LIN {X 0,Y 364.12,Z 423.241,A -85,B 0,C 180,E1 -13065.677,E2 -13065.677} C_VEL
LIN {X 0,Y 365.365,Z 412.607,A -85,B 0,C 180,E1 -13066.914,E2 -13066.914} C_VEL
LIN {X 0,Y 366.671,Z 400.866,A -85,B 0,C 180,E1 -13068.003,E2 -13068.003} C_VEL
LIN {X 0,Y 367.855,Z 388.491,A -85,B 0,C 180,E1 -13068.88,E2 -13068.88} C_VEL
LIN {X 0,Y 368.998,Z 374.969,A -85,B 0,C 180,E1 -13069.578,E2 -13069.578} C_VEL
LIN {X 0,Y 369.706,Z 361.353,A -85,B 0,C 180,E1 -13070.041,E2 -13070.041} C_VEL
LIN {X 0,Y 371.251,Z 294.99,A -85,B 0,C 180,E1 -13071.529,E2 -13071.529} C_VEL
LIN {X 0,Y 368.499,Z 273.063,A -85,B 0,C 180,E1 -13072.273,E2 -13072.273} C_VEL
LIN {X 0,Y 365.195,Z 254.41,A -85,B 0,C 180,E1 -13073,E2 -13073} C_VEL
LIN {X 0,Y 364.953,Z 252.892,A -85,B 0,C 180,E1 -13073.063,E2 -13073.063} C_VEL
LIN {X 0,Y 366.552,Z 235.571,A -85,B 0,C 180,E1 -13076.473,E2 -13076.473} C_VEL
LIN {X 0,Y 366.814,Z 231.096,A -85,B 0,C 180,E1 -13077.376,E2 -13077.376} C_VEL
LIN {X 0,Y 364.611,Z 220.318,A -85,B 0,C 180,E1 -13079.843,E2 -13079.843} C_VEL
LIN {X 0,Y 361.857,Z 209.412,A -85,B 0,C 180,E1 -13082.53,E2 -13082.53} C_VEL
LIN {X 0,Y 361.868,Z 209.408,A -85,B 0,C 180,E1 -13085.636,E2 -13085.636} C_VEL
LIN {X 0,Y 361.826,Z 209.413,A -85,B 0,C 180,E1 -13089.018,E2 -13089.018} C_VEL
LIN {X 0,Y 361.833,Z 209.411,A -85,B 0,C 180,E1 -13092.829,E2 -13092.829} C_VEL
LIN {X 0,Y 361.818,Z 209.413,A -85,B 0,C 180,E1 -13095.946,E2 -13095.946} C_VEL
LIN {X 0,Y 361.812,Z 209.413,A -85,B 0,C 180,E1 -13099.249,E2 -13099.249} C_VEL
LIN {X 0,Y 361.864,Z 209.41,A -85,B 0,C 180,E1 -13102.981,E2 -13102.981} C_VEL
LIN {X 0,Y 361.859,Z 209.41,A -85,B 0,C 180,E1 -13106.63,E2 -13106.63} C_VEL
LIN {X 0,Y 361.864,Z 209.409,A -85,B 0,C 180,E1 -13109.671,E2 -13109.671} C_VEL
LIN {X 0,Y 361.879,Z 209.403,A -85,B 0,C 180,E1 -13113.469,E2 -13113.469} C_VEL
LIN {X 0,Y 361.878,Z 209.404,A -85,B 0,C 180,E1 -13117.144,E2 -13117.144} C_VEL
LIN {X 0,Y 361.904,Z 209.404,A -85,B 0,C 180,E1 -13120.723,E2 -13120.723} C_VEL
LIN {X 0,Y 361.943,Z 209.399,A -85,B 0,C 180,E1 -13124.226,E2 -13124.226} C_VEL
LIN {X 0,Y 361.999,Z 209.391,A -85,B 0,C 180,E1 -13126.528,E2 -13126.528} C_VEL
LIN {X 0,Y 362.031,Z 209.388,A -85,B 0,C 180,E1 -13129.938,E2 -13129.938} C_VEL
LIN {X 0,Y 362.161,Z 209.372,A -85,B 0,C 180,E1 -13133.314,E2 -13133.314} C_VEL
LIN {X 0,Y 362.28,Z 209.358,A -85,B 0,C 180,E1 -13137.776,E2 -13137.776} C_VEL
LIN {X 0,Y 362.426,Z 209.34,A -85,B 0,C 180,E1 -13140,E2 -13140} C_VEL
LIN {X 0,Y 362.281,Z 209.358,A -85,B 0,C 180,E1 -13142.223,E2 -13142.223} C_VEL
LIN {X 0,Y 362.136,Z 209.375,A -85,B 0,C 180,E1 -13146.687,E2 -13146.687} C_VEL
LIN {X 0,Y 362,Z 209.395,A -85,B 0,C 180,E1 -13150.063,E2 -13150.063} C_VEL
LIN {X 0,Y 361.994,Z 209.4,A -85,B 0,C 180,E1 -13153.896,E2 -13153.896} C_VEL
LIN {X 0,Y 361.974,Z 209.407,A -85,B 0,C 180,E1 -13154.764,E2 -13154.764} C_VEL
LIN {X 0,Y 362.969,Z 212.239,A -85,B 0,C 180,E1 -13154.925,E2 -13154.925} C_VEL
LIN {X 0,Y 369.935,Z 226.404,A -85,B 0,C 180,E1 -13155.872,E2 -13155.872} C_VEL
LIN {X 0,Y 372.694,Z 233.181,A -85,B 0,C 180,E1 -13156.255,E2 -13156.255} C_VEL
LIN {X 0,Y 370.526,Z 315.426,A -85,B 0,C 180,E1 -13158.117,E2 -13158.117} C_VEL
LIN {X 0,Y 370.055,Z 328.234,A -85,B 0,C 180,E1 -13158.614,E2 -13158.614} C_VEL
LIN {X 0,Y 369.359,Z 340.587,A -85,B 0,C 180,E1 -13159.305,E2 -13159.305} C_VEL
LIN {X 0,Y 368.472,Z 352.076,A -85,B 0,C 180,E1 -13160.162,E2 -13160.162} C_VEL
LIN {X 0,Y 367.386,Z 363.949,A -85,B 0,C 180,E1 -13161.313,E2 -13161.313} C_VEL
LIN {X 0,Y 366.284,Z 374.257,A -85,B 0,C 180,E1 -13162.566,E2 -13162.566} C_VEL
LIN {X 0,Y 365.34,Z 382.674,A -85,B 0,C 180,E1 -13163.827,E2 -13163.827} C_VEL
LIN {X 0,Y 364.216,Z 391.354,A -85,B 0,C 180,E1 -13165.426,E2 -13165.426} C_VEL
LIN {X 0,Y 363.246,Z 398.749,A -85,B 0,C 180,E1 -13167.127,E2 -13167.127} C_VEL
LIN {X 0,Y 362.446,Z 405.12,A -85,B 0,C 180,E1 -13168.997,E2 -13168.997} C_VEL
LIN {X 0,Y 361.792,Z 409.737,A -85,B 0,C 180,E1 -13170.778,E2 -13170.778} C_VEL
LIN {X 0,Y 361.327,Z 412.797,A -85,B 0,C 180,E1 -13172.336,E2 -13172.336} C_VEL
LIN {X 0,Y 360.89,Z 415.46,A -85,B 0,C 180,E1 -13174.385,E2 -13174.385} C_VEL
LIN {X 0,Y 360.718,Z 416.5,A -85,B 0,C 180,E1 -13175.768,E2 -13175.768} C_VEL
LIN {X 0,Y 360.573,Z 416.872,A -85,B 0,C 180,E1 -13177.173,E2 -13177.173} C_VEL
LIN {X 0,Y 360.552,Z 416.539,A -85,B 0,C 180,E1 -13178.768,E2 -13178.768} C_VEL
LIN {X 0,Y 360.617,Z 415.206,A -85,B 0,C 180,E1 -13180.53,E2 -13180.53} C_VEL
LIN {X 0,Y 360.839,Z 412.887,A -85,B 0,C 180,E1 -13182.259,E2 -13182.259} C_VEL
LIN {X 0,Y 361.121,Z 409.624,A -85,B 0,C 180,E1 -13183.939,E2 -13183.939} C_VEL
LIN {X 0,Y 361.589,Z 404.185,A -85,B 0,C 180,E1 -13185.984,E2 -13185.984} C_VEL
LIN {X 0,Y 362.142,Z 397.638,A -85,B 0,C 180,E1 -13187.839,E2 -13187.839} C_VEL
LIN {X 0,Y 362.78,Z 390.677,A -85,B 0,C 180,E1 -13189.407,E2 -13189.407} C_VEL
LIN {X 0,Y 363.642,Z 381.431,A -85,B 0,C 180,E1 -13191.089,E2 -13191.089} C_VEL
LIN {X 0,Y 364.491,Z 372.167,A -85,B 0,C 180,E1 -13192.442,E2 -13192.442} C_VEL
LIN {X 0,Y 365.21,Z 361.929,A -85,B 0,C 180,E1 -13193.662,E2 -13193.662} C_VEL
LIN {X 0,Y 366.082,Z 350.464,A -85,B 0,C 180,E1 -13194.753,E2 -13194.753} C_VEL
LIN {X 0,Y 366.817,Z 339.184,A -85,B 0,C 180,E1 -13195.593,E2 -13195.593} C_VEL
LIN {X 0,Y 367.311,Z 325.985,A -85,B 0,C 180,E1 -13196.326,E2 -13196.326} C_VEL
LIN {X 0,Y 367.732,Z 313.177,A -85,B 0,C 180,E1 -13196.809,E2 -13196.809} C_VEL
LIN {X 0,Y 369.278,Z 229.303,A -85,B 0,C 180,E1 -13198.641,E2 -13198.641} C_VEL
LIN {X 0,Y 361.891,Z 209.408,A -85,B 0,C 180,E1 -13199.483,E2 -13199.483} C_VEL
LIN {X 0,Y 361.954,Z 209.398,A -85,B 0,C 180,E1 -13203.475,E2 -13203.475} C_VEL
LIN {X 0,Y 361.879,Z 209.41,A -85,B 0,C 180,E1 -13207.144,E2 -13207.144} C_VEL
LIN {X 0,Y 361.904,Z 209.405,A -85,B 0,C 180,E1 -13210.724,E2 -13210.724} C_VEL
LIN {X 0,Y 361.944,Z 209.397,A -85,B 0,C 180,E1 -13214.226,E2 -13214.226} C_VEL
LIN {X 0,Y 362,Z 209.392,A -85,B 0,C 180,E1 -13216.528,E2 -13216.528} C_VEL
LIN {X 0,Y 362.001,Z 209.389,A -85,B 0,C 180,E1 -13219.937,E2 -13219.937} C_VEL
LIN {X 0,Y 362.136,Z 209.373,A -85,B 0,C 180,E1 -13223.313,E2 -13223.313} C_VEL
LIN {X 0,Y 362.279,Z 209.355,A -85,B 0,C 180,E1 -13227.777,E2 -13227.777} C_VEL
LIN {X 0,Y 362.403,Z 209.341,A -85,B 0,C 180,E1 -13230,E2 -13230} C_VEL
LIN {X 0,Y 362.272,Z 209.359,A -85,B 0,C 180,E1 -13232.224,E2 -13232.224} C_VEL
LIN {X 0,Y 362.137,Z 209.375,A -85,B 0,C 180,E1 -13236.687,E2 -13236.687} C_VEL
LIN {X 0,Y 362.03,Z 209.39,A -85,B 0,C 180,E1 -13240.062,E2 -13240.062} C_VEL
LIN {X 0,Y 362,Z 209.393,A -85,B 0,C 180,E1 -13243.899,E2 -13243.899} C_VEL
LIN {X 0,Y 361.966,Z 209.395,A -85,B 0,C 180,E1 -13244.51,E2 -13244.51} C_VEL
LIN {X 0,Y 361.284,Z 209.481,A -85,B 0,C 180,E1 -13245.439,E2 -13245.439} C_VEL
LIN {X 0,Y 358.405,Z 209.837,A -85,B 0,C 180,E1 -13246.949,E2 -13246.949} C_VEL
LIN {X 0,Y 355.974,Z 210.145,A -85,B 0,C 180,E1 -13248.17,E2 -13248.17} C_VEL
LIN {X 0,Y 354.938,Z 210.27,A -85,B 0,C 180,E1 -13249.116,E2 -13249.116} C_VEL
LIN {X 0,Y 354.857,Z 210.28,A -85,B 0,C 180,E1 -13249.436,E2 -13249.436} C_VEL
LIN {X 0,Y 354.827,Z 210.284,A -85,B 0,C 180,E1 -13253.337,E2 -13253.337} C_VEL
LIN {X 0,Y 354.815,Z 210.284,A -85,B 0,C 180,E1 -13256.958,E2 -13256.958} C_VEL
LIN {X 0,Y 354.801,Z 210.291,A -85,B 0,C 180,E1 -13259.684,E2 -13259.684} C_VEL
LIN {X 0,Y 354.833,Z 210.288,A -85,B 0,C 180,E1 -13263.682,E2 -13263.682} C_VEL
LIN {X 0,Y 354.797,Z 210.287,A -85,B 0,C 180,E1 -13266.46,E2 -13266.46} C_VEL
LIN {X 0,Y 354.8,Z 210.291,A -85,B 0,C 180,E1 -13269.419,E2 -13269.419} C_VEL
LIN {X 0,Y 354.788,Z 210.289,A -85,B 0,C 180,E1 -13272.867,E2 -13272.867} C_VEL
LIN {X 0,Y 354.768,Z 210.291,A -85,B 0,C 180,E1 -13276.104,E2 -13276.104} C_VEL
LIN {X 0,Y 354.768,Z 210.295,A -85,B 0,C 180,E1 -13279.176,E2 -13279.176} C_VEL
LIN {X 0,Y 354.802,Z 210.286,A -85,B 0,C 180,E1 -13282.404,E2 -13282.404} C_VEL
LIN {X 0,Y 354.814,Z 210.288,A -85,B 0,C 180,E1 -13284.941,E2 -13284.941} C_VEL
LIN {X 0,Y 354.795,Z 210.287,A -85,B 0,C 180,E1 -13288.405,E2 -13288.405} C_VEL
LIN {X 0,Y 354.802,Z 210.287,A -85,B 0,C 180,E1 -13291.615,E2 -13291.615} C_VEL
LIN {X 0,Y 354.837,Z 210.282,A -85,B 0,C 180,E1 -13295.657,E2 -13295.657} C_VEL
LIN {X 0,Y 354.829,Z 210.286,A -85,B 0,C 180,E1 -13299.113,E2 -13299.113} C_VEL
LIN {X 0,Y 354.883,Z 210.282,A -85,B 0,C 180,E1 -13302.719,E2 -13302.719} C_VEL
LIN {X 0,Y 354.955,Z 210.269,A -85,B 0,C 180,E1 -13306.255,E2 -13306.255} C_VEL
LIN {X 0,Y 354.959,Z 210.266,A -85,B 0,C 180,E1 -13309.735,E2 -13309.735} C_VEL
LIN {X 0,Y 355.092,Z 210.251,A -85,B 0,C 180,E1 -13313.18,E2 -13313.18} C_VEL
LIN {X 0,Y 355.237,Z 210.232,A -85,B 0,C 180,E1 -13317.732,E2 -13317.732} C_VEL
LIN {X 0,Y 355.172,Z 210.24,A -85,B 0,C 180,E1 -13321.134,E2 -13321.134} C_VEL
LIN {X 0,Y 355.23,Z 210.238,A -85,B 0,C 180,E1 -13322.268,E2 -13322.268} C_VEL
LIN {X 0,Y 355.091,Z 210.251,A -85,B 0,C 180,E1 -13326.82,E2 -13326.82} C_VEL
LIN {X 0,Y 354.978,Z 210.269,A -85,B 0,C 180,E1 -13330.264,E2 -13330.264} C_VEL
LIN {X 0,Y 354.927,Z 210.277,A -85,B 0,C 180,E1 -13334.006,E2 -13334.006} C_VEL
LIN {X 0,Y 354.893,Z 210.279,A -85,B 0,C 180,E1 -13338.092,E2 -13338.092} C_VEL
LIN {X 0,Y 354.81,Z 210.288,A -85,B 0,C 180,E1 -13342.108,E2 -13342.108} C_VEL
LIN {X 0,Y 354.805,Z 210.291,A -85,B 0,C 180,E1 -13345.835,E2 -13345.835} C_VEL
LIN {X 0,Y 354.799,Z 210.292,A -85,B 0,C 180,E1 -13349.684,E2 -13349.684} C_VEL
LIN {X 0,Y 354.789,Z 210.288,A -85,B 0,C 180,E1 -13352.333,E2 -13352.333} C_VEL
LIN {X 0,Y 354.824,Z 210.287,A -85,B 0,C 180,E1 -13355.699,E2 -13355.699} C_VEL
LIN {X 0,Y 354.77,Z 210.296,A -85,B 0,C 180,E1 -13359.412,E2 -13359.412} C_VEL
LIN {X 0,Y 354.785,Z 210.29,A -85,B 0,C 180,E1 -13362.866,E2 -13362.866} C_VEL
LIN {X 0,Y 354.765,Z 210.291,A -85,B 0,C 180,E1 -13366.103,E2 -13366.103} C_VEL
LIN {X 0,Y 354.768,Z 210.296,A -85,B 0,C 180,E1 -13369.176,E2 -13369.176} C_VEL
LIN {X 0,Y 354.802,Z 210.286,A -85,B 0,C 180,E1 -13372.404,E2 -13372.404} C_VEL
LIN {X 0,Y 354.811,Z 210.29,A -85,B 0,C 180,E1 -13374.94,E2 -13374.94} C_VEL
LIN {X 0,Y 354.862,Z 210.35,A -85,B 0,C 180,E1 -13378.184,E2 -13378.184} C_VEL
LIN {X 0,Y 357.978,Z 224.948,A -85,B 0,C 180,E1 -13381.569,E2 -13381.569} C_VEL
LIN {X 0,Y 359.099,Z 232.517,A -85,B 0,C 180,E1 -13383.247,E2 -13383.247} C_VEL
LIN {X 0,Y 357.436,Z 250.02,A -85,B 0,C 180,E1 -13386.843,E2 -13386.843} C_VEL
LIN {X 0,Y 356.945,Z 256.387,A -85,B 0,C 180,E1 -13388.146,E2 -13388.146} C_VEL
LIN {X 0,Y 361.731,Z 295.758,A -85,B 0,C 180,E1 -13389.316,E2 -13389.316} C_VEL
LIN {X 0,Y 360.427,Z 366.272,A -85,B 0,C 180,E1 -13390.9,E2 -13390.9} C_VEL
LIN {X 0,Y 359.711,Z 379.611,A -85,B 0,C 180,E1 -13391.415,E2 -13391.415} C_VEL
LIN {X 0,Y 358.842,Z 391.905,A -85,B 0,C 180,E1 -13392.106,E2 -13392.106} C_VEL
LIN {X 0,Y 357.877,Z 403.805,A -85,B 0,C 180,E1 -13393.015,E2 -13393.015} C_VEL
LIN {X 0,Y 356.784,Z 415.28,A -85,B 0,C 180,E1 -13394.138,E2 -13394.138} C_VEL
LIN {X 0,Y 355.801,Z 425.857,A -85,B 0,C 180,E1 -13395.439,E2 -13395.439} C_VEL
LIN {X 0,Y 355.053,Z 435.016,A -85,B 0,C 180,E1 -13396.842,E2 -13396.842} C_VEL
LIN {X 0,Y 354.318,Z 444.104,A -85,B 0,C 180,E1 -13398.559,E2 -13398.559} C_VEL
LIN {X 0,Y 353.805,Z 451.39,A -85,B 0,C 180,E1 -13400.279,E2 -13400.279} C_VEL
LIN {X 0,Y 353.547,Z 457.173,A -85,B 0,C 180,E1 -13402.001,E2 -13402.001} C_VEL
LIN {X 0,Y 353.478,Z 461.845,A -85,B 0,C 180,E1 -13403.787,E2 -13403.787} C_VEL
LIN {X 0,Y 353.467,Z 465.089,A -85,B 0,C 180,E1 -13405.438,E2 -13405.438} C_VEL
LIN {X 0,Y 353.463,Z 466.749,A -85,B 0,C 180,E1 -13406.58,E2 -13406.58} C_VEL
LIN {X 0,Y 353.601,Z 467.995,A -85,B 0,C 180,E1 -13407.722,E2 -13407.722} C_VEL
LIN {X 0,Y 353.587,Z 468.794,A -85,B 0,C 180,E1 -13408.861,E2 -13408.861} C_VEL
LIN {X 0,Y 353.601,Z 469.137,A -85,B 0,C 180,E1 -13410,E2 -13410} C_VEL
LIN {X 0,Y 353.565,Z 469.067,A -85,B 0,C 180,E1 -13411.139,E2 -13411.139} C_VEL
LIN {X 0,Y 353.563,Z 468.594,A -85,B 0,C 180,E1 -13412.278,E2 -13412.278} C_VEL
LIN {X 0,Y 353.415,Z 467.681,A -85,B 0,C 180,E1 -13413.42,E2 -13413.42} C_VEL
LIN {X 0,Y 353.413,Z 466.325,A -85,B 0,C 180,E1 -13414.562,E2 -13414.562} C_VEL
LIN {X 0,Y 353.325,Z 464.08,A -85,B 0,C 180,E1 -13415.981,E2 -13415.981} C_VEL
LIN {X 0,Y 353.527,Z 459.629,A -85,B 0,C 180,E1 -13417.999,E2 -13417.999} C_VEL
LIN {X 0,Y 353.82,Z 454.623,A -85,B 0,C 180,E1 -13419.72,E2 -13419.72} C_VEL
LIN {X 0,Y 354.365,Z 448.345,A -85,B 0,C 180,E1 -13421.439,E2 -13421.439} C_VEL
LIN {X 0,Y 355.3,Z 440.578,A -85,B 0,C 180,E1 -13423.148,E2 -13423.148} C_VEL
LIN {X 0,Y 356.222,Z 432.29,A -85,B 0,C 180,E1 -13424.639,E2 -13424.639} C_VEL
LIN {X 0,Y 357.404,Z 422.065,A -85,B 0,C 180,E1 -13426.126,E2 -13426.126} C_VEL
LIN {X 0,Y 358.759,Z 411.304,A -85,B 0,C 180,E1 -13427.382,E2 -13427.382} C_VEL
LIN {X 0,Y 360.087,Z 399.395,A -85,B 0,C 180,E1 -13428.491,E2 -13428.491} C_VEL
LIN {X 0,Y 361.386,Z 386.803,A -85,B 0,C 180,E1 -13429.379,E2 -13429.379} C_VEL
LIN {X 0,Y 362.523,Z 373.725,A -85,B 0,C 180,E1 -13430.053,E2 -13430.053} C_VEL
LIN {X 0,Y 363.226,Z 360.002,A -85,B 0,C 180,E1 -13430.518,E2 -13430.518} C_VEL
LIN {X 0,Y 364.786,Z 295.309,A -85,B 0,C 180,E1 -13432,E2 -13432} C_VEL
LIN {X 0,Y 362.036,Z 273.374,A -85,B 0,C 180,E1 -13432.767,E2 -13432.767} C_VEL
LIN {X 0,Y 358.305,Z 252.123,A -85,B 0,C 180,E1 -13433.657,E2 -13433.657} C_VEL
LIN {X 0,Y 360.066,Z 234.037,A -85,B 0,C 180,E1 -13437.302,E2 -13437.302} C_VEL
LIN {X 0,Y 358.528,Z 225.173,A -85,B 0,C 180,E1 -13439.344,E2 -13439.344} C_VEL
LIN {X 0,Y 355.606,Z 213.37,A -85,B 0,C 180,E1 -13442.25,E2 -13442.25} C_VEL
LIN {X 0,Y 354.83,Z 210.287,A -85,B 0,C 180,E1 -13443.087,E2 -13443.087} C_VEL
LIN {X 0,Y 354.796,Z 210.291,A -85,B 0,C 180,E1 -13446.459,E2 -13446.459} C_VEL
LIN {X 0,Y 354.768,Z 210.292,A -85,B 0,C 180,E1 -13449.412,E2 -13449.412} C_VEL
LIN {X 0,Y 354.785,Z 210.288,A -85,B 0,C 180,E1 -13452.866,E2 -13452.866} C_VEL
LIN {X 0,Y 354.767,Z 210.292,A -85,B 0,C 180,E1 -13456.103,E2 -13456.103} C_VEL
LIN {X 0,Y 354.765,Z 210.291,A -85,B 0,C 180,E1 -13459.176,E2 -13459.176} C_VEL
LIN {X 0,Y 354.8,Z 210.287,A -85,B 0,C 180,E1 -13462.404,E2 -13462.404} C_VEL
LIN {X 0,Y 354.812,Z 210.284,A -85,B 0,C 180,E1 -13464.941,E2 -13464.941} C_VEL
LIN {X 0,Y 354.793,Z 210.289,A -85,B 0,C 180,E1 -13468.405,E2 -13468.405} C_VEL
LIN {X 0,Y 354.802,Z 210.287,A -85,B 0,C 180,E1 -13471.615,E2 -13471.615} C_VEL
LIN {X 0,Y 354.851,Z 210.283,A -85,B 0,C 180,E1 -13475.423,E2 -13475.423} C_VEL
LIN {X 0,Y 354.826,Z 210.283,A -85,B 0,C 180,E1 -13479.113,E2 -13479.113} C_VEL
LIN {X 0,Y 354.88,Z 210.274,A -85,B 0,C 180,E1 -13482.719,E2 -13482.719} C_VEL
LIN {X 0,Y 354.951,Z 210.27,A -85,B 0,C 180,E1 -13486.255,E2 -13486.255} C_VEL
LIN {X 0,Y 354.978,Z 210.269,A -85,B 0,C 180,E1 -13489.736,E2 -13489.736} C_VEL
LIN {X 0,Y 355.124,Z 210.249,A -85,B 0,C 180,E1 -13493.18,E2 -13493.18} C_VEL
LIN {X 0,Y 355.243,Z 210.235,A -85,B 0,C 180,E1 -13497.732,E2 -13497.732} C_VEL
LIN {X 0,Y 355.396,Z 210.216,A -85,B 0,C 180,E1 -13500,E2 -13500} C_VEL
LIN {X 0,Y 355.244,Z 210.235,A -85,B 0,C 180,E1 -13502.268,E2 -13502.268} C_VEL
LIN {X 0,Y 355.1,Z 210.252,A -85,B 0,C 180,E1 -13506.82,E2 -13506.82} C_VEL
LIN {X 0,Y 354.956,Z 210.273,A -85,B 0,C 180,E1 -13510.265,E2 -13510.265} C_VEL
LIN {X 0,Y 354.937,Z 210.277,A -85,B 0,C 180,E1 -13514.138,E2 -13514.138} C_VEL
LIN {X 0,Y 356.013,Z 213.217,A -85,B 0,C 180,E1 -13514.328,E2 -13514.328} C_VEL
LIN {X 0,Y 363.373,Z 228.03,A -85,B 0,C 180,E1 -13515.371,E2 -13515.371} C_VEL
LIN {X 0,Y 366.291,Z 234.841,A -85,B 0,C 180,E1 -13515.793,E2 -13515.793} C_VEL
LIN {X 0,Y 364.022,Z 316.501,A -85,B 0,C 180,E1 -13517.685,E2 -13517.685} C_VEL
LIN {X 0,Y 363.518,Z 329.543,A -85,B 0,C 180,E1 -13518.211,E2 -13518.211} C_VEL
LIN {X 0,Y 362.81,Z 341.52,A -85,B 0,C 180,E1 -13518.902,E2 -13518.902} C_VEL
LIN {X 0,Y 361.947,Z 352.263,A -85,B 0,C 180,E1 -13519.717,E2 -13519.717} C_VEL
LIN {X 0,Y 360.868,Z 363.435,A -85,B 0,C 180,E1 -13520.803,E2 -13520.803} C_VEL
LIN {X 0,Y 359.669,Z 374.037,A -85,B 0,C 180,E1 -13522.095,E2 -13522.095} C_VEL
LIN {X 0,Y 358.647,Z 382.574,A -85,B 0,C 180,E1 -13523.379,E2 -13523.379} C_VEL
LIN {X 0,Y 357.401,Z 391.803,A -85,B 0,C 180,E1 -13525.093,E2 -13525.093} C_VEL
LIN {X 0,Y 356.285,Z 399.819,A -85,B 0,C 180,E1 -13526.981,E2 -13526.981} C_VEL
LIN {X 0,Y 355.463,Z 406.042,A -85,B 0,C 180,E1 -13528.886,E2 -13528.886} C_VEL
LIN {X 0,Y 354.659,Z 411.236,A -85,B 0,C 180,E1 -13531.012,E2 -13531.012} C_VEL
LIN {X 0,Y 354.251,Z 413.699,A -85,B 0,C 180,E1 -13532.388,E2 -13532.388} C_VEL
LIN {X 0,Y 353.935,Z 415.555,A -85,B 0,C 180,E1 -13533.779,E2 -13533.779} C_VEL
LIN {X 0,Y 353.672,Z 416.914,A -85,B 0,C 180,E1 -13535.439,E2 -13535.439} C_VEL
LIN {X 0,Y 353.511,Z 417.425,A -85,B 0,C 180,E1 -13537.324,E2 -13537.324} C_VEL
LIN {X 0,Y 353.474,Z 416.61,A -85,B 0,C 180,E1 -13539.512,E2 -13539.512} C_VEL
LIN {X 0,Y 353.667,Z 414.238,A -85,B 0,C 180,E1 -13541.737,E2 -13541.737} C_VEL
LIN {X 0,Y 353.964,Z 411.566,A -85,B 0,C 180,E1 -13543.306,E2 -13543.306} C_VEL
LIN {X 0,Y 354.284,Z 407.887,A -85,B 0,C 180,E1 -13544.931,E2 -13544.931} C_VEL
LIN {X 0,Y 354.659,Z 403.179,A -85,B 0,C 180,E1 -13546.554,E2 -13546.554} C_VEL
LIN {X 0,Y 355.291,Z 396.245,A -85,B 0,C 180,E1 -13548.439,E2 -13548.439} C_VEL
LIN {X 0,Y 356.04,Z 388.374,A -85,B 0,C 180,E1 -13550.128,E2 -13550.128} C_VEL
LIN {X 0,Y 356.909,Z 378.998,A -85,B 0,C 180,E1 -13551.743,E2 -13551.743} C_VEL
LIN {X 0,Y 357.766,Z 369.571,A -85,B 0,C 180,E1 -13553.061,E2 -13553.061} C_VEL
LIN {X 0,Y 358.607,Z 358.616,A -85,B 0,C 180,E1 -13554.298,E2 -13554.298} C_VEL
LIN {X 0,Y 359.538,Z 346.218,A -85,B 0,C 180,E1 -13555.393,E2 -13555.393} C_VEL
LIN {X 0,Y 360.245,Z 333.921,A -85,B 0,C 180,E1 -13556.221,E2 -13556.221} C_VEL
LIN {X 0,Y 360.683,Z 321.379,A -85,B 0,C 180,E1 -13556.833,E2 -13556.833} C_VEL
LIN {X 0,Y 361.002,Z 307.837,A -85,B 0,C 180,E1 -13557.259,E2 -13557.259} C_VEL
LIN {X 0,Y 362.567,Z 230.978,A -85,B 0,C 180,E1 -13558.945,E2 -13558.945} C_VEL
LIN {X 0,Y 354.906,Z 210.542,A -85,B 0,C 180,E1 -13559.836,E2 -13559.836} C_VEL
LIN {X 0,Y 354.866,Z 210.279,A -85,B 0,C 180,E1 -13559.996,E2 -13559.996} C_VEL
LIN {X 0,Y 354.898,Z 210.274,A -85,B 0,C 180,E1 -13564.173,E2 -13564.173} C_VEL
LIN {X 0,Y 354.816,Z 210.284,A -85,B 0,C 180,E1 -13567.893,E2 -13567.893} C_VEL
LIN {X 0,Y 354.852,Z 210.281,A -85,B 0,C 180,E1 -13571.526,E2 -13571.526} C_VEL
LIN {X 0,Y 354.92,Z 210.275,A -85,B 0,C 180,E1 -13575.083,E2 -13575.083} C_VEL
LIN {X 0,Y 354.935,Z 210.273,A -85,B 0,C 180,E1 -13578.58,E2 -13578.58} C_VEL
LIN {X 0,Y 355.038,Z 210.257,A -85,B 0,C 180,E1 -13582.035,E2 -13582.035} C_VEL
LIN {X 0,Y 355.077,Z 210.255,A -85,B 0,C 180,E1 -13584.321,E2 -13584.321} C_VEL
LIN {X 0,Y 355.242,Z 210.231,A -85,B 0,C 180,E1 -13587.733,E2 -13587.733} C_VEL
LIN {X 0,Y 355.353,Z 210.219,A -85,B 0,C 180,E1 -13590,E2 -13590} C_VEL
LIN {X 0,Y 355.234,Z 210.236,A -85,B 0,C 180,E1 -13592.268,E2 -13592.268} C_VEL
LIN {X 0,Y 355.101,Z 210.25,A -85,B 0,C 180,E1 -13596.82,E2 -13596.82} C_VEL
LIN {X 0,Y 354.977,Z 210.27,A -85,B 0,C 180,E1 -13600.264,E2 -13600.264} C_VEL
LIN {X 0,Y 354.945,Z 210.273,A -85,B 0,C 180,E1 -13604.019,E2 -13604.019} C_VEL
LIN {X 0,Y 354.924,Z 210.277,A -85,B 0,C 180,E1 -13608.109,E2 -13608.109} C_VEL
LIN {X 0,Y 354.857,Z 210.28,A -85,B 0,C 180,E1 -13609.436,E2 -13609.436} C_VEL
LIN {X 0,Y 354.184,Z 210.369,A -85,B 0,C 180,E1 -13610.384,E2 -13610.384} C_VEL
LIN {X 0,Y 351.286,Z 210.731,A -85,B 0,C 180,E1 -13611.923,E2 -13611.923} C_VEL
LIN {X 0,Y 348.861,Z 211.031,A -85,B 0,C 180,E1 -13613.17,E2 -13613.17} C_VEL
LIN {X 0,Y 347.867,Z 211.154,A -85,B 0,C 180,E1 -13614.135,E2 -13614.135} C_VEL
LIN {X 0,Y 347.811,Z 211.158,A -85,B 0,C 180,E1 -13614.462,E2 -13614.462} C_VEL
LIN {X 0,Y 347.743,Z 211.17,A -85,B 0,C 180,E1 -13617.7,E2 -13617.7} C_VEL
LIN {X 0,Y 347.742,Z 211.167,A -85,B 0,C 180,E1 -13620.349,E2 -13620.349} C_VEL
LIN {X 0,Y 347.75,Z 211.167,A -85,B 0,C 180,E1 -13624.044,E2 -13624.044} C_VEL
LIN {X 0,Y 347.758,Z 211.167,A -85,B 0,C 180,E1 -13627.322,E2 -13627.322} C_VEL
LIN {X 0,Y 347.72,Z 211.169,A -85,B 0,C 180,E1 -13630.299,E2 -13630.299} C_VEL
LIN {X 0,Y 347.724,Z 211.173,A -85,B 0,C 180,E1 -13633.408,E2 -13633.408} C_VEL
LIN {X 0,Y 347.726,Z 211.168,A -85,B 0,C 180,E1 -13636.687,E2 -13636.687} C_VEL
LIN {X 0,Y 347.703,Z 211.17,A -85,B 0,C 180,E1 -13640.183,E2 -13640.183} C_VEL
LIN {X 0,Y 347.759,Z 211.165,A -85,B 0,C 180,E1 -13642.679,E2 -13642.679} C_VEL
LIN {X 0,Y 347.751,Z 211.165,A -85,B 0,C 180,E1 -13645.956,E2 -13645.956} C_VEL
LIN {X 0,Y 347.743,Z 211.166,A -85,B 0,C 180,E1 -13649.652,E2 -13649.652} C_VEL
LIN {X 0,Y 347.751,Z 211.165,A -85,B 0,C 180,E1 -13653.601,E2 -13653.601} C_VEL
LIN {X 0,Y 347.772,Z 211.162,A -85,B 0,C 180,E1 -13656.161,E2 -13656.161} C_VEL
LIN {X 0,Y 347.809,Z 211.157,A -85,B 0,C 180,E1 -13659.909,E2 -13659.909} C_VEL
LIN {X 0,Y 347.835,Z 211.154,A -85,B 0,C 180,E1 -13663.568,E2 -13663.568} C_VEL
LIN {X 0,Y 347.893,Z 211.148,A -85,B 0,C 180,E1 -13667.161,E2 -13667.161} C_VEL
LIN {X 0,Y 347.938,Z 211.146,A -85,B 0,C 180,E1 -13670.701,E2 -13670.701} C_VEL
LIN {X 0,Y 348.046,Z 211.131,A -85,B 0,C 180,E1 -13674.205,E2 -13674.205} C_VEL
LIN {X 0,Y 348.199,Z 211.109,A -85,B 0,C 180,E1 -13677.687,E2 -13677.687} C_VEL
LIN {X 0,Y 348.141,Z 211.116,A -85,B 0,C 180,E1 -13681.157,E2 -13681.157} C_VEL
LIN {X 0,Y 348.192,Z 211.116,A -85,B 0,C 180,E1 -13682.314,E2 -13682.314} C_VEL
LIN {X 0,Y 348.057,Z 211.126,A -85,B 0,C 180,E1 -13686.959,E2 -13686.959} C_VEL
LIN {X 0,Y 347.93,Z 211.145,A -85,B 0,C 180,E1 -13690.474,E2 -13690.474} C_VEL
LIN {X 0,Y 347.882,Z 211.153,A -85,B 0,C 180,E1 -13694.137,E2 -13694.137} C_VEL
LIN {X 0,Y 347.832,Z 211.157,A -85,B 0,C 180,E1 -13698.259,E2 -13698.259} C_VEL
LIN {X 0,Y 347.767,Z 211.166,A -85,B 0,C 180,E1 -13701.625,E2 -13701.625} C_VEL
LIN {X 0,Y 347.741,Z 211.166,A -85,B 0,C 180,E1 -13705.114,E2 -13705.114} C_VEL
LIN {X 0,Y 347.738,Z 211.172,A -85,B 0,C 180,E1 -13707.7,E2 -13707.7} C_VEL
LIN {X 0,Y 347.741,Z 211.166,A -85,B 0,C 180,E1 -13710.349,E2 -13710.349} C_VEL
LIN {X 0,Y 347.751,Z 211.166,A -85,B 0,C 180,E1 -13714.044,E2 -13714.044} C_VEL
LIN {X 0,Y 347.759,Z 211.168,A -85,B 0,C 180,E1 -13717.321,E2 -13717.321} C_VEL
LIN {X 0,Y 347.742,Z 211.169,A -85,B 0,C 180,E1 -13721.601,E2 -13721.601} C_VEL
LIN {X 0,Y 347.703,Z 211.174,A -85,B 0,C 180,E1 -13725.027,E2 -13725.027} C_VEL
LIN {X 0,Y 347.743,Z 211.165,A -85,B 0,C 180,E1 -13728.399,E2 -13728.399} C_VEL
LIN {X 0,Y 347.758,Z 211.165,A -85,B 0,C 180,E1 -13732.678,E2 -13732.678} C_VEL
LIN {X 0,Y 347.75,Z 211.166,A -85,B 0,C 180,E1 -13735.956,E2 -13735.956} C_VEL
LIN {X 0,Y 347.79,Z 211.176,A -85,B 0,C 180,E1 -13737.866,E2 -13737.866} C_VEL
LIN {X 0,Y 350.563,Z 223.964,A -85,B 0,C 180,E1 -13740.911,E2 -13740.911} C_VEL
LIN {X 0,Y 351.976,Z 231.602,A -85,B 0,C 180,E1 -13742.661,E2 -13742.661} C_VEL
LIN {X 0,Y 351.891,Z 236.038,A -85,B 0,C 180,E1 -13743.616,E2 -13743.616} C_VEL
LIN {X 0,Y 350.166,Z 254.148,A -85,B 0,C 180,E1 -13747.405,E2 -13747.405} C_VEL
LIN {X 0,Y 350.029,Z 255.919,A -85,B 0,C 180,E1 -13747.775,E2 -13747.775} C_VEL
LIN {X 0,Y 354.953,Z 296.667,A -85,B 0,C 180,E1 -13749.007,E2 -13749.007} C_VEL
LIN {X 0,Y 353.586,Z 365.641,A -85,B 0,C 180,E1 -13750.591,E2 -13750.591} C_VEL
LIN {X 0,Y 352.828,Z 379.747,A -85,B 0,C 180,E1 -13751.151,E2 -13751.151} C_VEL
LIN {X 0,Y 351.88,Z 392.339,A -85,B 0,C 180,E1 -13751.891,E2 -13751.891} C_VEL
LIN {X 0,Y 350.899,Z 404.032,A -85,B 0,C 180,E1 -13752.817,E2 -13752.817} C_VEL
LIN {X 0,Y 349.787,Z 415.378,A -85,B 0,C 180,E1 -13753.962,E2 -13753.962} C_VEL
LIN {X 0,Y 348.749,Z 425.95,A -85,B 0,C 180,E1 -13755.308,E2 -13755.308} C_VEL
LIN {X 0,Y 348.111,Z 434.079,A -85,B 0,C 180,E1 -13756.575,E2 -13756.575} C_VEL
LIN {X 0,Y 347.336,Z 443.243,A -85,B 0,C 180,E1 -13758.326,E2 -13758.326} C_VEL
LIN {X 0,Y 346.745,Z 450.601,A -85,B 0,C 180,E1 -13760.079,E2 -13760.079} C_VEL
LIN {X 0,Y 346.488,Z 456.454,A -85,B 0,C 180,E1 -13761.837,E2 -13761.837} C_VEL
LIN {X 0,Y 346.402,Z 461.469,A -85,B 0,C 180,E1 -13763.796,E2 -13763.796} C_VEL
LIN {X 0,Y 346.402,Z 464.461,A -85,B 0,C 180,E1 -13765.345,E2 -13765.345} C_VEL
LIN {X 0,Y 346.376,Z 466.139,A -85,B 0,C 180,E1 -13766.51,E2 -13766.51} C_VEL
LIN {X 0,Y 346.534,Z 467.405,A -85,B 0,C 180,E1 -13767.675,E2 -13767.675} C_VEL
LIN {X 0,Y 346.52,Z 468.233,A -85,B 0,C 180,E1 -13768.838,E2 -13768.838} C_VEL
LIN {X 0,Y 346.53,Z 468.598,A -85,B 0,C 180,E1 -13770,E2 -13770} C_VEL
LIN {X 0,Y 346.499,Z 468.546,A -85,B 0,C 180,E1 -13771.162,E2 -13771.162} C_VEL
LIN {X 0,Y 346.479,Z 468.089,A -85,B 0,C 180,E1 -13772.325,E2 -13772.325} C_VEL
LIN {X 0,Y 346.327,Z 467.209,A -85,B 0,C 180,E1 -13773.49,E2 -13773.49} C_VEL
LIN {X 0,Y 346.315,Z 465.877,A -85,B 0,C 180,E1 -13774.656,E2 -13774.656} C_VEL
LIN {X 0,Y 346.242,Z 463.899,A -85,B 0,C 180,E1 -13775.956,E2 -13775.956} C_VEL
LIN {X 0,Y 346.402,Z 460.644,A -85,B 0,C 180,E1 -13777.578,E2 -13777.578} C_VEL
LIN {X 0,Y 346.648,Z 456.069,A -85,B 0,C 180,E1 -13779.334,E2 -13779.334} C_VEL
LIN {X 0,Y 347.115,Z 450.282,A -85,B 0,C 180,E1 -13781.089,E2 -13781.089} C_VEL
LIN {X 0,Y 348.036,Z 443.113,A -85,B 0,C 180,E1 -13782.834,E2 -13782.834} C_VEL
LIN {X 0,Y 349.004,Z 434.836,A -85,B 0,C 180,E1 -13784.465,E2 -13784.465} C_VEL
LIN {X 0,Y 350.155,Z 425.135,A -85,B 0,C 180,E1 -13786.02,E2 -13786.02} C_VEL
LIN {X 0,Y 351.658,Z 414.044,A -85,B 0,C 180,E1 -13787.444,E2 -13787.444} C_VEL
LIN {X 0,Y 353.071,Z 402.917,A -85,B 0,C 180,E1 -13788.571,E2 -13788.571} C_VEL
LIN {X 0,Y 354.422,Z 390.59,A -85,B 0,C 180,E1 -13789.549,E2 -13789.549} C_VEL
LIN {X 0,Y 355.642,Z 377.724,A -85,B 0,C 180,E1 -13790.307,E2 -13790.307} C_VEL
LIN {X 0,Y 356.615,Z 364.159,A -85,B 0,C 180,E1 -13790.85,E2 -13790.85} C_VEL
LIN {X 0,Y 357.723,Z 325.967,A -85,B 0,C 180,E1 -13791.766,E2 -13791.766} C_VEL
LIN {X 0,Y 358.404,Z 296.296,A -85,B 0,C 180,E1 -13792.469,E2 -13792.469} C_VEL
LIN {X 0,Y 355.88,Z 275.588,A -85,B 0,C 180,E1 -13793.221,E2 -13793.221} C_VEL
LIN {X 0,Y 352.618,Z 256.749,A -85,B 0,C 180,E1 -13794.007,E2 -13794.007} C_VEL
LIN {X 0,Y 351.623,Z 251.541,A -85,B 0,C 180,E1 -13794.251,E2 -13794.251} C_VEL
LIN {X 0,Y 353.297,Z 235.548,A -85,B 0,C 180,E1 -13797.548,E2 -13797.548} C_VEL
LIN {X 0,Y 351.677,Z 226.668,A -85,B 0,C 180,E1 -13799.643,E2 -13799.643} C_VEL
LIN {X 0,Y 348.929,Z 215.478,A -85,B 0,C 180,E1 -13802.479,E2 -13802.479} C_VEL
LIN {X 0,Y 347.794,Z 211.164,A -85,B 0,C 180,E1 -13803.635,E2 -13803.635} C_VEL
LIN {X 0,Y 347.757,Z 211.165,A -85,B 0,C 180,E1 -13807.321,E2 -13807.321} C_VEL
LIN {X 0,Y 347.741,Z 211.167,A -85,B 0,C 180,E1 -13811.601,E2 -13811.601} C_VEL
LIN {X 0,Y 347.705,Z 211.169,A -85,B 0,C 180,E1 -13815.027,E2 -13815.027} C_VEL
LIN {X 0,Y 347.741,Z 211.168,A -85,B 0,C 180,E1 -13818.399,E2 -13818.399} C_VEL
LIN {X 0,Y 347.756,Z 211.165,A -85,B 0,C 180,E1 -13822.678,E2 -13822.678} C_VEL
LIN {X 0,Y 347.748,Z 211.167,A -85,B 0,C 180,E1 -13825.956,E2 -13825.956} C_VEL
LIN {X 0,Y 347.74,Z 211.169,A -85,B 0,C 180,E1 -13829.651,E2 -13829.651} C_VEL
LIN {X 0,Y 347.758,Z 211.161,A -85,B 0,C 180,E1 -13833.602,E2 -13833.602} C_VEL
LIN {X 0,Y 347.77,Z 211.161,A -85,B 0,C 180,E1 -13836.16,E2 -13836.16} C_VEL
LIN {X 0,Y 347.805,Z 211.157,A -85,B 0,C 180,E1 -13839.909,E2 -13839.909} C_VEL
LIN {X 0,Y 347.832,Z 211.155,A -85,B 0,C 180,E1 -13843.568,E2 -13843.568} C_VEL
LIN {X 0,Y 347.89,Z 211.15,A -85,B 0,C 180,E1 -13847.16,E2 -13847.16} C_VEL
LIN {X 0,Y 347.944,Z 211.14,A -85,B 0,C 180,E1 -13850.701,E2 -13850.701} C_VEL
LIN {X 0,Y 348.09,Z 211.126,A -85,B 0,C 180,E1 -13853.042,E2 -13853.042} C_VEL
LIN {X 0,Y 348.205,Z 211.112,A -85,B 0,C 180,E1 -13857.686,E2 -13857.686} C_VEL
LIN {X 0,Y 348.345,Z 211.094,A -85,B 0,C 180,E1 -13860,E2 -13860} C_VEL
LIN {X 0,Y 348.206,Z 211.112,A -85,B 0,C 180,E1 -13862.313,E2 -13862.313} C_VEL
LIN {X 0,Y 348.068,Z 211.129,A -85,B 0,C 180,E1 -13866.958,E2 -13866.958} C_VEL
LIN {X 0,Y 347.896,Z 211.153,A -85,B 0,C 180,E1 -13870.475,E2 -13870.475} C_VEL
LIN {X 0,Y 347.884,Z 211.16,A -85,B 0,C 180,E1 -13873.471,E2 -13873.471} C_VEL
LIN {X 0,Y 349.015,Z 214.181,A -85,B 0,C 180,E1 -13873.686,E2 -13873.686} C_VEL
LIN {X 0,Y 355.902,Z 227.519,A -85,B 0,C 180,E1 -13874.705,E2 -13874.705} C_VEL
LIN {X 0,Y 359.963,Z 236.56,A -85,B 0,C 180,E1 -13875.302,E2 -13875.302} C_VEL
LIN {X 0,Y 357.527,Z 317.728,A -85,B 0,C 180,E1 -13877.241,E2 -13877.241} C_VEL
LIN {X 0,Y 357.015,Z 331.017,A -85,B 0,C 180,E1 -13877.803,E2 -13877.803} C_VEL
LIN {X 0,Y 356.283,Z 342.618,A -85,B 0,C 180,E1 -13878.496,E2 -13878.496} C_VEL
LIN {X 0,Y 355.335,Z 353.463,A -85,B 0,C 180,E1 -13879.344,E2 -13879.344} C_VEL
LIN {X 0,Y 354.214,Z 364.667,A -85,B 0,C 180,E1 -13880.469,E2 -13880.469} C_VEL
LIN {X 0,Y 353.006,Z 374.69,A -85,B 0,C 180,E1 -13881.719,E2 -13881.719} C_VEL
LIN {X 0,Y 351.771,Z 384.341,A -85,B 0,C 180,E1 -13883.216,E2 -13883.216} C_VEL
LIN {X 0,Y 350.503,Z 393.028,A -85,B 0,C 180,E1 -13884.902,E2 -13884.902} C_VEL
LIN {X 0,Y 349.486,Z 399.967,A -85,B 0,C 180,E1 -13886.579,E2 -13886.579} C_VEL
LIN {X 0,Y 348.692,Z 405.56,A -85,B 0,C 180,E1 -13888.271,E2 -13888.271} C_VEL
LIN {X 0,Y 347.847,Z 410.823,A -85,B 0,C 180,E1 -13890.338,E2 -13890.338} C_VEL
LIN {X 0,Y 347.364,Z 413.648,A -85,B 0,C 180,E1 -13891.815,E2 -13891.815} C_VEL
LIN {X 0,Y 346.867,Z 416.31,A -85,B 0,C 180,E1 -13893.828,E2 -13893.828} C_VEL
LIN {X 0,Y 346.523,Z 417.764,A -85,B 0,C 180,E1 -13896.027,E2 -13896.027} C_VEL
LIN {X 0,Y 346.41,Z 417.906,A -85,B 0,C 180,E1 -13897.699,E2 -13897.699} C_VEL
LIN {X 0,Y 346.392,Z 417.073,A -85,B 0,C 180,E1 -13899.558,E2 -13899.558} C_VEL
LIN {X 0,Y 346.53,Z 415.243,A -85,B 0,C 180,E1 -13901.375,E2 -13901.375} C_VEL
LIN {X 0,Y 346.924,Z 411.708,A -85,B 0,C 180,E1 -13903.533,E2 -13903.533} C_VEL
LIN {X 0,Y 347.26,Z 408.126,A -85,B 0,C 180,E1 -13905.1,E2 -13905.1} C_VEL
LIN {X 0,Y 347.765,Z 402.296,A -85,B 0,C 180,E1 -13907.079,E2 -13907.079} C_VEL
LIN {X 0,Y 348.316,Z 396.194,A -85,B 0,C 180,E1 -13908.705,E2 -13908.705} C_VEL
LIN {X 0,Y 349.055,Z 388.676,A -85,B 0,C 180,E1 -13910.327,E2 -13910.327} C_VEL
LIN {X 0,Y 349.932,Z 379.573,A -85,B 0,C 180,E1 -13911.922,E2 -13911.922} C_VEL
LIN {X 0,Y 350.87,Z 369.512,A -85,B 0,C 180,E1 -13913.351,E2 -13913.351} C_VEL
LIN {X 0,Y 351.744,Z 358.584,A -85,B 0,C 180,E1 -13914.59,E2 -13914.59} C_VEL
LIN {X 0,Y 352.666,Z 346.715,A -85,B 0,C 180,E1 -13915.652,E2 -13915.652} C_VEL
LIN {X 0,Y 353.328,Z 335.434,A -85,B 0,C 180,E1 -13916.437,E2 -13916.437} C_VEL
LIN {X 0,Y 353.767,Z 322.663,A -85,B 0,C 180,E1 -13917.09,E2 -13917.09} C_VEL
LIN {X 0,Y 354.158,Z 308.853,A -85,B 0,C 180,E1 -13917.542,E2 -13917.542} C_VEL
LIN {X 0,Y 355.782,Z 232.516,A -85,B 0,C 180,E1 -13919.261,E2 -13919.261} C_VEL
LIN {X 0,Y 347.821,Z 211.157,A -85,B 0,C 180,E1 -13920.217,E2 -13920.217} C_VEL
LIN {X 0,Y 347.83,Z 211.156,A -85,B 0,C 180,E1 -13923.608,E2 -13923.608} C_VEL
LIN {X 0,Y 347.785,Z 211.16,A -85,B 0,C 180,E1 -13926.162,E2 -13926.162} C_VEL
LIN {X 0,Y 347.806,Z 211.157,A -85,B 0,C 180,E1 -13929.909,E2 -13929.909} C_VEL
LIN {X 0,Y 347.833,Z 211.155,A -85,B 0,C 180,E1 -13933.569,E2 -13933.569} C_VEL
LIN {X 0,Y 347.891,Z 211.15,A -85,B 0,C 180,E1 -13937.161,E2 -13937.161} C_VEL
LIN {X 0,Y 347.936,Z 211.147,A -85,B 0,C 180,E1 -13940.701,E2 -13940.701} C_VEL
LIN {X 0,Y 348.051,Z 211.129,A -85,B 0,C 180,E1 -13944.206,E2 -13944.206} C_VEL
LIN {X 0,Y 348.204,Z 211.108,A -85,B 0,C 180,E1 -13947.687,E2 -13947.687} C_VEL
LIN {X 0,Y 348.304,Z 211.097,A -85,B 0,C 180,E1 -13950,E2 -13950} C_VEL
LIN {X 0,Y 348.196,Z 211.114,A -85,B 0,C 180,E1 -13952.314,E2 -13952.314} C_VEL
LIN {X 0,Y 348.069,Z 211.126,A -85,B 0,C 180,E1 -13956.959,E2 -13956.959} C_VEL
LIN {X 0,Y 347.929,Z 211.146,A -85,B 0,C 180,E1 -13960.475,E2 -13960.475} C_VEL
LIN {X 0,Y 347.9,Z 211.152,A -85,B 0,C 180,E1 -13964.15,E2 -13964.15} C_VEL
LIN {X 0,Y 347.893,Z 211.15,A -85,B 0,C 180,E1 -13968.291,E2 -13968.291} C_VEL
LIN {X 0,Y 347.769,Z 211.165,A -85,B 0,C 180,E1 -13971.627,E2 -13971.627} C_VEL
LIN {X 0,Y 347.811,Z 211.158,A -85,B 0,C 180,E1 -13974.462,E2 -13974.462} C_VEL
LIN {X 0,Y 347.187,Z 211.238,A -85,B 0,C 180,E1 -13975.428,E2 -13975.428} C_VEL
LIN {X 0,Y 344.272,Z 211.598,A -85,B 0,C 180,E1 -13976.998,E2 -13976.998} C_VEL
LIN {X 0,Y 341.792,Z 211.909,A -85,B 0,C 180,E1 -13978.27,E2 -13978.27} C_VEL
LIN {X 0,Y 340.764,Z 212.036,A -85,B 0,C 180,E1 -13979.255,E2 -13979.255} C_VEL
LIN {X 0,Y 340.703,Z 212.046,A -85,B 0,C 180,E1 -13979.589,E2 -13979.589} C_VEL
LIN {X 0,Y 340.691,Z 212.044,A -85,B 0,C 180,E1 -13982.436,E2 -13982.436} C_VEL
LIN {X 0,Y 340.719,Z 212.043,A -85,B 0,C 180,E1 -13985.279,E2 -13985.279} C_VEL
LIN {X 0,Y 340.695,Z 212.044,A -85,B 0,C 180,E1 -13988.383,E2 -13988.383} C_VEL
LIN {X 0,Y 340.698,Z 212.044,A -85,B 0,C 180,E1 -13992.045,E2 -13992.045} C_VEL
LIN {X 0,Y 340.653,Z 212.049,A -85,B 0,C 180,E1 -13996.227,E2 -13996.227} C_VEL
LIN {X 0,Y 340.673,Z 212.047,A -85,B 0,C 180,E1 -13998.688,E2 -13998.688} C_VEL
LIN {X 0,Y 340.721,Z 212.042,A -85,B 0,C 180,E1 -14001.771,E2 -14001.771} C_VEL
LIN {X 0,Y 340.725,Z 212.042,A -85,B 0,C 180,E1 -14005.596,E2 -14005.596} C_VEL
LIN {X 0,Y 340.697,Z 212.048,A -85,B 0,C 180,E1 -14008.955,E2 -14008.955} C_VEL
LIN {X 0,Y 340.722,Z 212.046,A -85,B 0,C 180,E1 -14013.013,E2 -14013.013} C_VEL
LIN {X 0,Y 340.744,Z 212.038,A -85,B 0,C 180,E1 -14015.637,E2 -14015.637} C_VEL
LIN {X 0,Y 340.736,Z 212.039,A -85,B 0,C 180,E1 -14019.474,E2 -14019.474} C_VEL
LIN {X 0,Y 340.795,Z 212.031,A -85,B 0,C 180,E1 -14021.981,E2 -14021.981} C_VEL
LIN {X 0,Y 340.873,Z 212.021,A -85,B 0,C 180,E1 -14025.705,E2 -14025.705} C_VEL
LIN {X 0,Y 340.851,Z 212.024,A -85,B 0,C 180,E1 -14029.306,E2 -14029.306} C_VEL
LIN {X 0,Y 341.006,Z 212.007,A -85,B 0,C 180,E1 -14032.897,E2 -14032.897} C_VEL
LIN {X 0,Y 340.828,Z 212.027,A -85,B 0,C 180,E1 -14035.269,E2 -14035.269} C_VEL
LIN {X 0,Y 341.16,Z 211.986,A -85,B 0,C 180,E1 -14037.639,E2 -14037.639} C_VEL
LIN {X 0,Y 341.11,Z 211.992,A -85,B 0,C 180,E1 -14041.181,E2 -14041.181} C_VEL
LIN {X 0,Y 341.129,Z 211.995,A -85,B 0,C 180,E1 -14042.362,E2 -14042.362} C_VEL
LIN {X 0,Y 341.018,Z 212.006,A -85,B 0,C 180,E1 -14045.915,E2 -14045.915} C_VEL
LIN {X 0,Y 340.914,Z 212.017,A -85,B 0,C 180,E1 -14049.493,E2 -14049.493} C_VEL
LIN {X 0,Y 340.845,Z 212.025,A -85,B 0,C 180,E1 -14053.11,E2 -14053.11} C_VEL
LIN {X 0,Y 340.753,Z 212.036,A -85,B 0,C 180,E1 -14056.783,E2 -14056.783} C_VEL
LIN {X 0,Y 340.761,Z 212.036,A -85,B 0,C 180,E1 -14059.268,E2 -14059.268} C_VEL
LIN {X 0,Y 340.704,Z 212.043,A -85,B 0,C 180,E1 -14063.075,E2 -14063.075} C_VEL
LIN {X 0,Y 340.72,Z 212.041,A -85,B 0,C 180,E1 -14066.987,E2 -14066.987} C_VEL
LIN {X 0,Y 340.696,Z 212.044,A -85,B 0,C 180,E1 -14071.045,E2 -14071.045} C_VEL
LIN {X 0,Y 340.72,Z 212.044,A -85,B 0,C 180,E1 -14075.279,E2 -14075.279} C_VEL
LIN {X 0,Y 340.696,Z 212.043,A -85,B 0,C 180,E1 -14078.382,E2 -14078.382} C_VEL
LIN {X 0,Y 340.694,Z 212.044,A -85,B 0,C 180,E1 -14082.044,E2 -14082.044} C_VEL
LIN {X 0,Y 340.652,Z 212.049,A -85,B 0,C 180,E1 -14086.227,E2 -14086.227} C_VEL
LIN {X 0,Y 340.673,Z 212.047,A -85,B 0,C 180,E1 -14088.688,E2 -14088.688} C_VEL
LIN {X 0,Y 340.721,Z 212.041,A -85,B 0,C 180,E1 -14091.771,E2 -14091.771} C_VEL
LIN {X 0,Y 340.724,Z 212.043,A -85,B 0,C 180,E1 -14095.596,E2 -14095.596} C_VEL
LIN {X 0,Y 340.755,Z 212.108,A -85,B 0,C 180,E1 -14097.571,E2 -14097.571} C_VEL
LIN {X 0,Y 343.683,Z 225.688,A -85,B 0,C 180,E1 -14100.868,E2 -14100.868} C_VEL
LIN {X 0,Y 345.095,Z 233.66,A -85,B 0,C 180,E1 -14102.727,E2 -14102.727} C_VEL
LIN {X 0,Y 344.105,Z 245.37,A -85,B 0,C 180,E1 -14105.248,E2 -14105.248} C_VEL
LIN {X 0,Y 343.122,Z 255.458,A -85,B 0,C 180,E1 -14107.395,E2 -14107.395} C_VEL
LIN {X 0,Y 348.159,Z 297.319,A -85,B 0,C 180,E1 -14108.693,E2 -14108.693} C_VEL
LIN {X 0,Y 346.719,Z 365.705,A -85,B 0,C 180,E1 -14110.306,E2 -14110.306} C_VEL
LIN {X 0,Y 345.924,Z 379.61,A -85,B 0,C 180,E1 -14110.876,E2 -14110.876} C_VEL
LIN {X 0,Y 345.023,Z 391.588,A -85,B 0,C 180,E1 -14111.595,E2 -14111.595} C_VEL
LIN {X 0,Y 343.911,Z 404.114,A -85,B 0,C 180,E1 -14112.61,E2 -14112.61} C_VEL
LIN {X 0,Y 342.792,Z 415.358,A -85,B 0,C 180,E1 -14113.779,E2 -14113.779} C_VEL
LIN {X 0,Y 341.696,Z 425.955,A -85,B 0,C 180,E1 -14115.172,E2 -14115.172} C_VEL
LIN {X 0,Y 340.966,Z 434.709,A -85,B 0,C 180,E1 -14116.592,E2 -14116.592} C_VEL
LIN {X 0,Y 340.185,Z 443.684,A -85,B 0,C 180,E1 -14118.379,E2 -14118.379} C_VEL
LIN {X 0,Y 339.645,Z 450.823,A -85,B 0,C 180,E1 -14120.171,E2 -14120.171} C_VEL
LIN {X 0,Y 339.371,Z 457.343,A -85,B 0,C 180,E1 -14122.264,E2 -14122.264} C_VEL
LIN {X 0,Y 339.299,Z 461.587,A -85,B 0,C 180,E1 -14124.055,E2 -14124.055} C_VEL
LIN {X 0,Y 339.335,Z 463.807,A -85,B 0,C 180,E1 -14125.248,E2 -14125.248} C_VEL
LIN {X 0,Y 339.292,Z 465.508,A -85,B 0,C 180,E1 -14126.437,E2 -14126.437} C_VEL
LIN {X 0,Y 339.467,Z 466.799,A -85,B 0,C 180,E1 -14127.627,E2 -14127.627} C_VEL
LIN {X 0,Y 339.454,Z 467.654,A -85,B 0,C 180,E1 -14128.813,E2 -14128.813} C_VEL
LIN {X 0,Y 339.462,Z 468.058,A -85,B 0,C 180,E1 -14130,E2 -14130} C_VEL
LIN {X 0,Y 339.433,Z 468.026,A -85,B 0,C 180,E1 -14131.186,E2 -14131.186} C_VEL
LIN {X 0,Y 339.38,Z 467.585,A -85,B 0,C 180,E1 -14132.373,E2 -14132.373} C_VEL
LIN {X 0,Y 339.241,Z 466.732,A -85,B 0,C 180,E1 -14133.563,E2 -14133.563} C_VEL
LIN {X 0,Y 339.221,Z 465.43,A -85,B 0,C 180,E1 -14134.753,E2 -14134.753} C_VEL
LIN {X 0,Y 339.197,Z 462.676,A -85,B 0,C 180,E1 -14136.543,E2 -14136.543} C_VEL
LIN {X 0,Y 339.402,Z 458.885,A -85,B 0,C 180,E1 -14138.334,E2 -14138.334} C_VEL
LIN {X 0,Y 339.723,Z 453.962,A -85,B 0,C 180,E1 -14140.127,E2 -14140.127} C_VEL
LIN {X 0,Y 340.418,Z 447.794,A -85,B 0,C 180,E1 -14141.914,E2 -14141.914} C_VEL
LIN {X 0,Y 341.386,Z 440.159,A -85,B 0,C 180,E1 -14143.694,E2 -14143.694} C_VEL
LIN {X 0,Y 342.594,Z 430.735,A -85,B 0,C 180,E1 -14145.467,E2 -14145.467} C_VEL
LIN {X 0,Y 343.94,Z 421.006,A -85,B 0,C 180,E1 -14146.928,E2 -14146.928} C_VEL
LIN {X 0,Y 345.422,Z 410.289,A -85,B 0,C 180,E1 -14148.229,E2 -14148.229} C_VEL
LIN {X 0,Y 346.907,Z 398.418,A -85,B 0,C 180,E1 -14149.374,E2 -14149.374} C_VEL
LIN {X 0,Y 348.353,Z 385.869,A -85,B 0,C 180,E1 -14150.289,E2 -14150.289} C_VEL
LIN {X 0,Y 349.535,Z 372.939,A -85,B 0,C 180,E1 -14150.986,E2 -14150.986} C_VEL
LIN {X 0,Y 350.277,Z 360.61,A -85,B 0,C 180,E1 -14151.441,E2 -14151.441} C_VEL
LIN {X 0,Y 352.076,Z 297.228,A -85,B 0,C 180,E1 -14152.968,E2 -14152.968} C_VEL
LIN {X 0,Y 349.447,Z 275.565,A -85,B 0,C 180,E1 -14153.78,E2 -14153.78} C_VEL
LIN {X 0,Y 345.845,Z 255.264,A -85,B 0,C 180,E1 -14154.674,E2 -14154.674} C_VEL
LIN {X 0,Y 345.003,Z 250.877,A -85,B 0,C 180,E1 -14154.892,E2 -14154.892} C_VEL
LIN {X 0,Y 346.501,Z 237.059,A -85,B 0,C 180,E1 -14157.807,E2 -14157.807} C_VEL
LIN {X 0,Y 344.537,Z 226.777,A -85,B 0,C 180,E1 -14160.322,E2 -14160.322} C_VEL
LIN {X 0,Y 341.899,Z 216.352,A -85,B 0,C 180,E1 -14163.063,E2 -14163.063} C_VEL
LIN {X 0,Y 340.717,Z 212.046,A -85,B 0,C 180,E1 -14164.292,E2 -14164.292} C_VEL
LIN {X 0,Y 340.719,Z 212.044,A -85,B 0,C 180,E1 -14168.229,E2 -14168.229} C_VEL
LIN {X 0,Y 340.693,Z 212.046,A -85,B 0,C 180,E1 -14172.044,E2 -14172.044} C_VEL
LIN {X 0,Y 340.651,Z 212.051,A -85,B 0,C 180,E1 -14176.227,E2 -14176.227} C_VEL
LIN {X 0,Y 340.671,Z 212.05,A -85,B 0,C 180,E1 -14178.688,E2 -14178.688} C_VEL
LIN {X 0,Y 340.719,Z 212.043,A -85,B 0,C 180,E1 -14181.77,E2 -14181.77} C_VEL
LIN {X 0,Y 340.723,Z 212.04,A -85,B 0,C 180,E1 -14185.595,E2 -14185.595} C_VEL
LIN {X 0,Y 340.694,Z 212.046,A -85,B 0,C 180,E1 -14188.955,E2 -14188.955} C_VEL
LIN {X 0,Y 340.725,Z 212.038,A -85,B 0,C 180,E1 -14193.013,E2 -14193.013} C_VEL
LIN {X 0,Y 340.754,Z 212.039,A -85,B 0,C 180,E1 -14195.638,E2 -14195.638} C_VEL
LIN {X 0,Y 340.733,Z 212.037,A -85,B 0,C 180,E1 -14199.473,E2 -14199.473} C_VEL
LIN {X 0,Y 340.792,Z 212.031,A -85,B 0,C 180,E1 -14201.981,E2 -14201.981} C_VEL
LIN {X 0,Y 340.869,Z 212.02,A -85,B 0,C 180,E1 -14205.705,E2 -14205.705} C_VEL
LIN {X 0,Y 340.871,Z 212.022,A -85,B 0,C 180,E1 -14209.306,E2 -14209.306} C_VEL
LIN {X 0,Y 341.058,Z 212.001,A -85,B 0,C 180,E1 -14212.898,E2 -14212.898} C_VEL
LIN {X 0,Y 341.167,Z 211.989,A -85,B 0,C 180,E1 -14217.639,E2 -14217.639} C_VEL
LIN {X 0,Y 341.295,Z 211.972,A -85,B 0,C 180,E1 -14220,E2 -14220} C_VEL
LIN {X 0,Y 341.168,Z 211.988,A -85,B 0,C 180,E1 -14222.361,E2 -14222.361} C_VEL
LIN {X 0,Y 341.037,Z 212.006,A -85,B 0,C 180,E1 -14227.103,E2 -14227.103} C_VEL
LIN {X 0,Y 340.848,Z 212.031,A -85,B 0,C 180,E1 -14230.694,E2 -14230.694} C_VEL
LIN {X 0,Y 340.851,Z 212.034,A -85,B 0,C 180,E1 -14232.768,E2 -14232.768} C_VEL
LIN {X 0,Y 341.927,Z 214.979,A -85,B 0,C 180,E1 -14232.992,E2 -14232.992} C_VEL
LIN {X 0,Y 345.035,Z 220.588,A -85,B 0,C 180,E1 -14233.471,E2 -14233.471} C_VEL
LIN {X 0,Y 352.296,Z 235.445,A -85,B 0,C 180,E1 -14234.593,E2 -14234.593} C_VEL
LIN {X 0,Y 353.688,Z 238.654,A -85,B 0,C 180,E1 -14234.805,E2 -14234.805} C_VEL
LIN {X 0,Y 351.172,Z 317.971,A -85,B 0,C 180,E1 -14236.735,E2 -14236.735} C_VEL
LIN {X 0,Y 350.617,Z 331.407,A -85,B 0,C 180,E1 -14237.312,E2 -14237.312} C_VEL
LIN {X 0,Y 349.799,Z 343.732,A -85,B 0,C 180,E1 -14238.069,E2 -14238.069} C_VEL
LIN {X 0,Y 348.589,Z 356.158,A -85,B 0,C 180,E1 -14239.094,E2 -14239.094} C_VEL
LIN {X 0,Y 347.417,Z 367.05,A -85,B 0,C 180,E1 -14240.252,E2 -14240.252} C_VEL
LIN {X 0,Y 346.112,Z 377.192,A -85,B 0,C 180,E1 -14241.595,E2 -14241.595} C_VEL
LIN {X 0,Y 344.876,Z 386.231,A -85,B 0,C 180,E1 -14243.083,E2 -14243.083} C_VEL
LIN {X 0,Y 343.583,Z 394.655,A -85,B 0,C 180,E1 -14244.792,E2 -14244.792} C_VEL
LIN {X 0,Y 342.5,Z 401.463,A -85,B 0,C 180,E1 -14246.519,E2 -14246.519} C_VEL
LIN {X 0,Y 341.688,Z 406.831,A -85,B 0,C 180,E1 -14248.234,E2 -14248.234} C_VEL
LIN {X 0,Y 340.749,Z 412.161,A -85,B 0,C 180,E1 -14250.483,E2 -14250.483} C_VEL
LIN {X 0,Y 340.115,Z 415.507,A -85,B 0,C 180,E1 -14252.497,E2 -14252.497} C_VEL
LIN {X 0,Y 339.72,Z 417.291,A -85,B 0,C 180,E1 -14254.157,E2 -14254.157} C_VEL
LIN {X 0,Y 339.452,Z 418.384,A -85,B 0,C 180,E1 -14256.153,E2 -14256.153} C_VEL
LIN {X 0,Y 339.313,Z 418.224,A -85,B 0,C 180,E1 -14258.416,E2 -14258.416} C_VEL
LIN {X 0,Y 339.324,Z 417.256,A -85,B 0,C 180,E1 -14259.974,E2 -14259.974} C_VEL
LIN {X 0,Y 339.517,Z 415.169,A -85,B 0,C 180,E1 -14261.824,E2 -14261.824} C_VEL
LIN {X 0,Y 339.873,Z 412.096,A -85,B 0,C 180,E1 -14263.636,E2 -14263.636} C_VEL
LIN {X 0,Y 340.257,Z 408.077,A -85,B 0,C 180,E1 -14265.391,E2 -14265.391} C_VEL
LIN {X 0,Y 340.816,Z 401.869,A -85,B 0,C 180,E1 -14267.455,E2 -14267.455} C_VEL
LIN {X 0,Y 341.41,Z 395.478,A -85,B 0,C 180,E1 -14269.129,E2 -14269.129} C_VEL
LIN {X 0,Y 342.309,Z 387.153,A -85,B 0,C 180,E1 -14270.887,E2 -14270.887} C_VEL
LIN {X 0,Y 343.086,Z 378.963,A -85,B 0,C 180,E1 -14272.3,E2 -14272.3} C_VEL
LIN {X 0,Y 344.013,Z 369.27,A -85,B 0,C 180,E1 -14273.669,E2 -14273.669} C_VEL
LIN {X 0,Y 344.932,Z 358.058,A -85,B 0,C 180,E1 -14274.943,E2 -14274.943} C_VEL
LIN {X 0,Y 345.901,Z 346.12,A -85,B 0,C 180,E1 -14276.01,E2 -14276.01} C_VEL
LIN {X 0,Y 346.639,Z 332.983,A -85,B 0,C 180,E1 -14276.892,E2 -14276.892} C_VEL
LIN {X 0,Y 347.055,Z 320.795,A -85,B 0,C 180,E1 -14277.484,E2 -14277.484} C_VEL
LIN {X 0,Y 347.405,Z 307.091,A -85,B 0,C 180,E1 -14277.903,E2 -14277.903} C_VEL
LIN {X 0,Y 349.076,Z 234.356,A -85,B 0,C 180,E1 -14279.571,E2 -14279.571} C_VEL
LIN {X 0,Y 340.803,Z 212.094,A -85,B 0,C 180,E1 -14280.59,E2 -14280.59} C_VEL
LIN {X 0,Y 340.772,Z 212.034,A -85,B 0,C 180,E1 -14284.336,E2 -14284.336} C_VEL
LIN {X 0,Y 340.742,Z 212.038,A -85,B 0,C 180,E1 -14288.207,E2 -14288.207} C_VEL
LIN {X 0,Y 340.793,Z 212.031,A -85,B 0,C 180,E1 -14291.981,E2 -14291.981} C_VEL
LIN {X 0,Y 340.87,Z 212.022,A -85,B 0,C 180,E1 -14295.705,E2 -14295.705} C_VEL
LIN {X 0,Y 340.849,Z 212.025,A -85,B 0,C 180,E1 -14299.306,E2 -14299.306} C_VEL
LIN {X 0,Y 341.01,Z 212.008,A -85,B 0,C 180,E1 -14302.897,E2 -14302.897} C_VEL
LIN {X 0,Y 340.833,Z 212.027,A -85,B 0,C 180,E1 -14305.269,E2 -14305.269} C_VEL
LIN {X 0,Y 341.166,Z 211.985,A -85,B 0,C 180,E1 -14307.639,E2 -14307.639} C_VEL
LIN {X 0,Y 341.256,Z 211.975,A -85,B 0,C 180,E1 -14310,E2 -14310} C_VEL
LIN {X 0,Y 341.157,Z 211.991,A -85,B 0,C 180,E1 -14312.362,E2 -14312.362} C_VEL
LIN {X 0,Y 341.017,Z 212.003,A -85,B 0,C 180,E1 -14317.103,E2 -14317.103} C_VEL
LIN {X 0,Y 340.871,Z 212.023,A -85,B 0,C 180,E1 -14320.694,E2 -14320.694} C_VEL
LIN {X 0,Y 340.865,Z 212.026,A -85,B 0,C 180,E1 -14324.325,E2 -14324.325} C_VEL
LIN {X 0,Y 340.839,Z 212.028,A -85,B 0,C 180,E1 -14328.467,E2 -14328.467} C_VEL
LIN {X 0,Y 340.719,Z 212.045,A -85,B 0,C 180,E1 -14331.842,E2 -14331.842} C_VEL
LIN {X 0,Y 340.738,Z 212.042,A -85,B 0,C 180,E1 -14335.668,E2 -14335.668} C_VEL
LIN {X 0,Y 340.703,Z 212.046,A -85,B 0,C 180,E1 -14339.589,E2 -14339.589} C_VEL
LIN {X 0,Y 340.105,Z 212.128,A -85,B 0,C 180,E1 -14340.576,E2 -14340.576} C_VEL
LIN {X 0,Y 337.302,Z 212.48,A -85,B 0,C 180,E1 -14342.182,E2 -14342.182} C_VEL
LIN {X 0,Y 334.866,Z 212.778,A -85,B 0,C 180,E1 -14343.482,E2 -14343.482} C_VEL
LIN {X 0,Y 333.787,Z 212.906,A -85,B 0,C 180,E1 -14344.488,E2 -14344.488} C_VEL
LIN {X 0,Y 333.683,Z 212.916,A -85,B 0,C 180,E1 -14344.829,E2 -14344.829} C_VEL
LIN {X 0,Y 333.645,Z 212.927,A -85,B 0,C 180,E1 -14347.653,E2 -14347.653} C_VEL
LIN {X 0,Y 333.644,Z 212.922,A -85,B 0,C 180,E1 -14350.768,E2 -14350.768} C_VEL
LIN {X 0,Y 333.595,Z 212.928,A -85,B 0,C 180,E1 -14354.251,E2 -14354.251} C_VEL
LIN {X 0,Y 333.64,Z 212.926,A -85,B 0,C 180,E1 -14357.618,E2 -14357.618} C_VEL
LIN {X 0,Y 333.636,Z 212.928,A -85,B 0,C 180,E1 -14361.206,E2 -14361.206} C_VEL
LIN {X 0,Y 333.677,Z 212.918,A -85,B 0,C 180,E1 -14363.861,E2 -14363.861} C_VEL
LIN {X 0,Y 333.646,Z 212.925,A -85,B 0,C 180,E1 -14367.413,E2 -14367.413} C_VEL
LIN {X 0,Y 333.657,Z 212.926,A -85,B 0,C 180,E1 -14371.023,E2 -14371.023} C_VEL
LIN {X 0,Y 333.699,Z 212.919,A -85,B 0,C 180,E1 -14375.089,E2 -14375.089} C_VEL
LIN {X 0,Y 333.676,Z 212.922,A -85,B 0,C 180,E1 -14379.019,E2 -14379.019} C_VEL
LIN {X 0,Y 333.744,Z 212.909,A -85,B 0,C 180,E1 -14381.587,E2 -14381.587} C_VEL
LIN {X 0,Y 333.811,Z 212.901,A -85,B 0,C 180,E1 -14385.577,E2 -14385.577} C_VEL
LIN {X 0,Y 333.821,Z 212.901,A -85,B 0,C 180,E1 -14389.078,E2 -14389.078} C_VEL
LIN {X 0,Y 333.961,Z 212.886,A -85,B 0,C 180,E1 -14392.746,E2 -14392.746} C_VEL
LIN {X 0,Y 333.794,Z 212.904,A -85,B 0,C 180,E1 -14395.169,E2 -14395.169} C_VEL
LIN {X 0,Y 334.097,Z 212.865,A -85,B 0,C 180,E1 -14397.589,E2 -14397.589} C_VEL
LIN {X 0,Y 334.079,Z 212.868,A -85,B 0,C 180,E1 -14401.206,E2 -14401.206} C_VEL
LIN {X 0,Y 334.069,Z 212.874,A -85,B 0,C 180,E1 -14402.412,E2 -14402.412} C_VEL
LIN {X 0,Y 333.992,Z 212.882,A -85,B 0,C 180,E1 -14406.039,E2 -14406.039} C_VEL
LIN {X 0,Y 333.851,Z 212.898,A -85,B 0,C 180,E1 -14409.696,E2 -14409.696} C_VEL
LIN {X 0,Y 333.79,Z 212.904,A -85,B 0,C 180,E1 -14413.392,E2 -14413.392} C_VEL
LIN {X 0,Y 333.703,Z 212.915,A -85,B 0,C 180,E1 -14417.149,E2 -14417.149} C_VEL
LIN {X 0,Y 333.687,Z 212.92,A -85,B 0,C 180,E1 -14419.693,E2 -14419.693} C_VEL
LIN {X 0,Y 333.645,Z 212.925,A -85,B 0,C 180,E1 -14423.592,E2 -14423.592} C_VEL
LIN {X 0,Y 333.669,Z 212.923,A -85,B 0,C 180,E1 -14427.606,E2 -14427.606} C_VEL
LIN {X 0,Y 333.66,Z 212.92,A -85,B 0,C 180,E1 -14430.366,E2 -14430.366} C_VEL
LIN {X 0,Y 333.64,Z 212.925,A -85,B 0,C 180,E1 -14433.208,E2 -14433.208} C_VEL
LIN {X 0,Y 333.677,Z 212.918,A -85,B 0,C 180,E1 -14436.139,E2 -14436.139} C_VEL
LIN {X 0,Y 333.622,Z 212.928,A -85,B 0,C 180,E1 -14439.196,E2 -14439.196} C_VEL
LIN {X 0,Y 333.629,Z 212.924,A -85,B 0,C 180,E1 -14442.499,E2 -14442.499} C_VEL
LIN {X 0,Y 333.596,Z 212.928,A -85,B 0,C 180,E1 -14445.954,E2 -14445.954} C_VEL
LIN {X 0,Y 333.604,Z 212.931,A -85,B 0,C 180,E1 -14449.324,E2 -14449.324} C_VEL
LIN {X 0,Y 333.664,Z 212.924,A -85,B 0,C 180,E1 -14453.168,E2 -14453.168} C_VEL
LIN {X 0,Y 333.675,Z 212.922,A -85,B 0,C 180,E1 -14456.795,E2 -14456.795} C_VEL
LIN {X 0,Y 333.743,Z 213.109,A -85,B 0,C 180,E1 -14457.287,E2 -14457.287} C_VEL
LIN {X 0,Y 336.592,Z 226.459,A -85,B 0,C 180,E1 -14460.6,E2 -14460.6} C_VEL
LIN {X 0,Y 338.067,Z 234.187,A -85,B 0,C 180,E1 -14462.448,E2 -14462.448} C_VEL
LIN {X 0,Y 337.749,Z 240.049,A -85,B 0,C 180,E1 -14463.751,E2 -14463.751} C_VEL
LIN {X 0,Y 336.213,Z 254.949,A -85,B 0,C 180,E1 -14466.994,E2 -14466.994} C_VEL
LIN {X 0,Y 341.354,Z 297.764,A -85,B 0,C 180,E1 -14468.363,E2 -14468.363} C_VEL
LIN {X 0,Y 339.866,Z 364.672,A -85,B 0,C 180,E1 -14469.971,E2 -14469.971} C_VEL
LIN {X 0,Y 339.043,Z 378.721,A -85,B 0,C 180,E1 -14470.551,E2 -14470.551} C_VEL
LIN {X 0,Y 338.181,Z 390.833,A -85,B 0,C 180,E1 -14471.287,E2 -14471.287} C_VEL
LIN {X 0,Y 337.133,Z 402.622,A -85,B 0,C 180,E1 -14472.249,E2 -14472.249} C_VEL
LIN {X 0,Y 335.876,Z 414.024,A -85,B 0,C 180,E1 -14473.435,E2 -14473.435} C_VEL
LIN {X 0,Y 334.829,Z 424.367,A -85,B 0,C 180,E1 -14474.789,E2 -14474.789} C_VEL
LIN {X 0,Y 334.029,Z 433.687,A -85,B 0,C 180,E1 -14476.308,E2 -14476.308} C_VEL
LIN {X 0,Y 333.206,Z 442.75,A -85,B 0,C 180,E1 -14478.132,E2 -14478.132} C_VEL
LIN {X 0,Y 332.586,Z 449.992,A -85,B 0,C 180,E1 -14479.96,E2 -14479.96} C_VEL
LIN {X 0,Y 332.337,Z 454.893,A -85,B 0,C 180,E1 -14481.487,E2 -14481.487} C_VEL
LIN {X 0,Y 332.225,Z 459.736,A -85,B 0,C 180,E1 -14483.379,E2 -14483.379} C_VEL
LIN {X 0,Y 332.268,Z 463.142,A -85,B 0,C 180,E1 -14485.146,E2 -14485.146} C_VEL
LIN {X 0,Y 332.211,Z 464.878,A -85,B 0,C 180,E1 -14486.361,E2 -14486.361} C_VEL
LIN {X 0,Y 332.382,Z 466.191,A -85,B 0,C 180,E1 -14487.576,E2 -14487.576} C_VEL
LIN {X 0,Y 332.391,Z 467.071,A -85,B 0,C 180,E1 -14488.788,E2 -14488.788} C_VEL
LIN {X 0,Y 332.395,Z 467.517,A -85,B 0,C 180,E1 -14490,E2 -14490} C_VEL
LIN {X 0,Y 332.369,Z 467.505,A -85,B 0,C 180,E1 -14491.211,E2 -14491.211} C_VEL
LIN {X 0,Y 332.283,Z 467.08,A -85,B 0,C 180,E1 -14492.424,E2 -14492.424} C_VEL
LIN {X 0,Y 332.158,Z 466.248,A -85,B 0,C 180,E1 -14493.639,E2 -14493.639} C_VEL
LIN {X 0,Y 332.131,Z 464.983,A -85,B 0,C 180,E1 -14494.855,E2 -14494.855} C_VEL
LIN {X 0,Y 332.117,Z 462.274,A -85,B 0,C 180,E1 -14496.683,E2 -14496.683} C_VEL
LIN {X 0,Y 332.329,Z 458.535,A -85,B 0,C 180,E1 -14498.513,E2 -14498.513} C_VEL
LIN {X 0,Y 332.689,Z 453.677,A -85,B 0,C 180,E1 -14500.344,E2 -14500.344} C_VEL
LIN {X 0,Y 333.46,Z 447.567,A -85,B 0,C 180,E1 -14502.167,E2 -14502.167} C_VEL
LIN {X 0,Y 334.438,Z 439.99,A -85,B 0,C 180,E1 -14503.985,E2 -14503.985} C_VEL
LIN {X 0,Y 335.74,Z 430.651,A -85,B 0,C 180,E1 -14505.791,E2 -14505.791} C_VEL
LIN {X 0,Y 337.154,Z 421.037,A -85,B 0,C 180,E1 -14507.28,E2 -14507.28} C_VEL
LIN {X 0,Y 338.694,Z 410.485,A -85,B 0,C 180,E1 -14508.604,E2 -14508.604} C_VEL
LIN {X 0,Y 340.252,Z 398.873,A -85,B 0,C 180,E1 -14509.769,E2 -14509.769} C_VEL
LIN {X 0,Y 341.729,Z 386.749,A -85,B 0,C 180,E1 -14510.7,E2 -14510.7} C_VEL
LIN {X 0,Y 343.092,Z 372.868,A -85,B 0,C 180,E1 -14511.478,E2 -14511.478} C_VEL
LIN {X 0,Y 343.915,Z 359.671,A -85,B 0,C 180,E1 -14511.976,E2 -14511.976} C_VEL
LIN {X 0,Y 345.754,Z 297.928,A -85,B 0,C 180,E1 -14513.496,E2 -14513.496} C_VEL
LIN {X 0,Y 343.258,Z 276.937,A -85,B 0,C 180,E1 -14514.309,E2 -14514.309} C_VEL
LIN {X 0,Y 339.45,Z 255.406,A -85,B 0,C 180,E1 -14515.3,E2 -14515.3} C_VEL
LIN {X 0,Y 338.447,Z 250.204,A -85,B 0,C 180,E1 -14515.57,E2 -14515.57} C_VEL
LIN {X 0,Y 339.714,Z 238.6,A -85,B 0,C 180,E1 -14518.076,E2 -14518.076} C_VEL
LIN {X 0,Y 337.756,Z 228.558,A -85,B 0,C 180,E1 -14520.604,E2 -14520.604} C_VEL
LIN {X 0,Y 335.149,Z 218.287,A -85,B 0,C 180,E1 -14523.397,E2 -14523.397} C_VEL
LIN {X 0,Y 333.666,Z 212.925,A -85,B 0,C 180,E1 -14524.94,E2 -14524.94} C_VEL
LIN {X 0,Y 333.643,Z 212.924,A -85,B 0,C 180,E1 -14527.652,E2 -14527.652} C_VEL
LIN {X 0,Y 333.603,Z 212.927,A -85,B 0,C 180,E1 -14530.774,E2 -14530.774} C_VEL
LIN {X 0,Y 333.593,Z 212.931,A -85,B 0,C 180,E1 -14534.25,E2 -14534.25} C_VEL
LIN {X 0,Y 333.638,Z 212.92,A -85,B 0,C 180,E1 -14537.618,E2 -14537.618} C_VEL
LIN {X 0,Y 333.634,Z 212.926,A -85,B 0,C 180,E1 -14541.206,E2 -14541.206} C_VEL
LIN {X 0,Y 333.675,Z 212.922,A -85,B 0,C 180,E1 -14543.861,E2 -14543.861} C_VEL
LIN {X 0,Y 333.645,Z 212.921,A -85,B 0,C 180,E1 -14547.412,E2 -14547.412} C_VEL
LIN {X 0,Y 333.655,Z 212.92,A -85,B 0,C 180,E1 -14551.022,E2 -14551.022} C_VEL
LIN {X 0,Y 333.708,Z 212.916,A -85,B 0,C 180,E1 -14555.089,E2 -14555.089} C_VEL
LIN {X 0,Y 333.672,Z 212.918,A -85,B 0,C 180,E1 -14559.019,E2 -14559.019} C_VEL
LIN {X 0,Y 333.741,Z 212.913,A -85,B 0,C 180,E1 -14561.586,E2 -14561.586} C_VEL
LIN {X 0,Y 333.808,Z 212.9,A -85,B 0,C 180,E1 -14565.577,E2 -14565.577} C_VEL
LIN {X 0,Y 333.833,Z 212.898,A -85,B 0,C 180,E1 -14569.078,E2 -14569.078} C_VEL
LIN {X 0,Y 334.006,Z 212.88,A -85,B 0,C 180,E1 -14572.747,E2 -14572.747} C_VEL
LIN {X 0,Y 333.807,Z 212.906,A -85,B 0,C 180,E1 -14575.169,E2 -14575.169} C_VEL
LIN {X 0,Y 334.104,Z 212.869,A -85,B 0,C 180,E1 -14577.589,E2 -14577.589} C_VEL
LIN {X 0,Y 334.246,Z 212.851,A -85,B 0,C 180,E1 -14580,E2 -14580} C_VEL
LIN {X 0,Y 334.105,Z 212.868,A -85,B 0,C 180,E1 -14582.411,E2 -14582.411} C_VEL
LIN {X 0,Y 333.978,Z 212.882,A -85,B 0,C 180,E1 -14586.492,E2 -14586.492} C_VEL
LIN {X 0,Y 333.82,Z 212.906,A -85,B 0,C 180,E1 -14589.696,E2 -14589.696} C_VEL
LIN {X 0,Y 333.807,Z 212.91,A -85,B 0,C 180,E1 -14592.038,E2 -14592.038} C_VEL
LIN {X 0,Y 334.888,Z 215.9,A -85,B 0,C 180,E1 -14592.256,E2 -14592.256} C_VEL
LIN {X 0,Y 338.014,Z 221.39,A -85,B 0,C 180,E1 -14592.769,E2 -14592.769} C_VEL
LIN {X 0,Y 345.282,Z 235.699,A -85,B 0,C 180,E1 -14593.93,E2 -14593.93} C_VEL
LIN {X 0,Y 347.412,Z 240.513,A -85,B 0,C 180,E1 -14594.275,E2 -14594.275} C_VEL
LIN {X 0,Y 344.832,Z 318.782,A -85,B 0,C 180,E1 -14596.232,E2 -14596.232} C_VEL
LIN {X 0,Y 344.254,Z 331.767,A -85,B 0,C 180,E1 -14596.798,E2 -14596.798} C_VEL
LIN {X 0,Y 343.378,Z 344.208,A -85,B 0,C 180,E1 -14597.571,E2 -14597.571} C_VEL
LIN {X 0,Y 342.13,Z 356.706,A -85,B 0,C 180,E1 -14598.62,E2 -14598.62} C_VEL
LIN {X 0,Y 340.806,Z 368.393,A -85,B 0,C 180,E1 -14599.893,E2 -14599.893} C_VEL
LIN {X 0,Y 339.392,Z 378.456,A -85,B 0,C 180,E1 -14601.277,E2 -14601.277} C_VEL
LIN {X 0,Y 337.952,Z 388.195,A -85,B 0,C 180,E1 -14602.95,E2 -14602.95} C_VEL
LIN {X 0,Y 336.639,Z 396.254,A -85,B 0,C 180,E1 -14604.679,E2 -14604.679} C_VEL
LIN {X 0,Y 335.534,Z 402.793,A -85,B 0,C 180,E1 -14606.43,E2 -14606.43} C_VEL
LIN {X 0,Y 334.518,Z 408.745,A -85,B 0,C 180,E1 -14608.461,E2 -14608.461} C_VEL
LIN {X 0,Y 333.749,Z 412.957,A -85,B 0,C 180,E1 -14610.357,E2 -14610.357} C_VEL
LIN {X 0,Y 333.076,Z 416.251,A -85,B 0,C 180,E1 -14612.434,E2 -14612.434} C_VEL
LIN {X 0,Y 332.538,Z 418.405,A -85,B 0,C 180,E1 -14614.794,E2 -14614.794} C_VEL
LIN {X 0,Y 332.333,Z 419.011,A -85,B 0,C 180,E1 -14616.525,E2 -14616.525} C_VEL
LIN {X 0,Y 332.227,Z 418.687,A -85,B 0,C 180,E1 -14618.491,E2 -14618.491} C_VEL
LIN {X 0,Y 332.32,Z 416.777,A -85,B 0,C 180,E1 -14620.965,E2 -14620.965} C_VEL
LIN {X 0,Y 332.718,Z 413.251,A -85,B 0,C 180,E1 -14623.328,E2 -14623.328} C_VEL
LIN {X 0,Y 333.168,Z 408.766,A -85,B 0,C 180,E1 -14625.393,E2 -14625.393} C_VEL
LIN {X 0,Y 333.757,Z 402.692,A -85,B 0,C 180,E1 -14627.477,E2 -14627.477} C_VEL
LIN {X 0,Y 334.425,Z 395.685,A -85,B 0,C 180,E1 -14629.348,E2 -14629.348} C_VEL
LIN {X 0,Y 335.394,Z 386.764,A -85,B 0,C 180,E1 -14631.244,E2 -14631.244} C_VEL
LIN {X 0,Y 336.397,Z 376.943,A -85,B 0,C 180,E1 -14632.897,E2 -14632.897} C_VEL
LIN {X 0,Y 337.356,Z 366.348,A -85,B 0,C 180,E1 -14634.338,E2 -14634.338} C_VEL
LIN {X 0,Y 338.325,Z 355.356,A -85,B 0,C 180,E1 -14635.524,E2 -14635.524} C_VEL
LIN {X 0,Y 339.285,Z 342.326,A -85,B 0,C 180,E1 -14636.618,E2 -14636.618} C_VEL
LIN {X 0,Y 339.94,Z 329.437,A -85,B 0,C 180,E1 -14637.419,E2 -14637.419} C_VEL
LIN {X 0,Y 340.364,Z 317.156,A -85,B 0,C 180,E1 -14637.95,E2 -14637.95} C_VEL
LIN {X 0,Y 340.861,Z 296.364,A -85,B 0,C 180,E1 -14638.485,E2 -14638.485} C_VEL
LIN {X 0,Y 342.309,Z 235.901,A -85,B 0,C 180,E1 -14639.904,E2 -14639.904} C_VEL
LIN {X 0,Y 333.731,Z 212.916,A -85,B 0,C 180,E1 -14640.987,E2 -14640.987} C_VEL
LIN {X 0,Y 333.718,Z 212.916,A -85,B 0,C 180,E1 -14644.9,E2 -14644.9} C_VEL
LIN {X 0,Y 333.674,Z 212.924,A -85,B 0,C 180,E1 -14649.019,E2 -14649.019} C_VEL
LIN {X 0,Y 333.742,Z 212.91,A -85,B 0,C 180,E1 -14651.587,E2 -14651.587} C_VEL
LIN {X 0,Y 333.809,Z 212.902,A -85,B 0,C 180,E1 -14655.577,E2 -14655.577} C_VEL
LIN {X 0,Y 333.819,Z 212.903,A -85,B 0,C 180,E1 -14659.078,E2 -14659.078} C_VEL
LIN {X 0,Y 333.964,Z 212.887,A -85,B 0,C 180,E1 -14662.746,E2 -14662.746} C_VEL
LIN {X 0,Y 333.798,Z 212.904,A -85,B 0,C 180,E1 -14665.169,E2 -14665.169} C_VEL
LIN {X 0,Y 334.103,Z 212.865,A -85,B 0,C 180,E1 -14667.589,E2 -14667.589} C_VEL
LIN {X 0,Y 334.208,Z 212.853,A -85,B 0,C 180,E1 -14670,E2 -14670} C_VEL
LIN {X 0,Y 334.094,Z 212.871,A -85,B 0,C 180,E1 -14672.412,E2 -14672.412} C_VEL
LIN {X 0,Y 333.999,Z 212.88,A -85,B 0,C 180,E1 -14676.04,E2 -14676.04} C_VEL
LIN {X 0,Y 333.85,Z 212.897,A -85,B 0,C 180,E1 -14679.696,E2 -14679.696} C_VEL
LIN {X 0,Y 333.798,Z 212.903,A -85,B 0,C 180,E1 -14683.392,E2 -14683.392} C_VEL
LIN {X 0,Y 333.748,Z 212.909,A -85,B 0,C 180,E1 -14687.146,E2 -14687.146} C_VEL
LIN {X 0,Y 333.735,Z 212.913,A -85,B 0,C 180,E1 -14689.691,E2 -14689.691} C_VEL
LIN {X 0,Y 333.669,Z 212.921,A -85,B 0,C 180,E1 -14693.591,E2 -14693.591} C_VEL
LIN {X 0,Y 333.669,Z 212.921,A -85,B 0,C 180,E1 -14696.252,E2 -14696.252} C_VEL
LIN {X 0,Y 333.659,Z 212.921,A -85,B 0,C 180,E1 -14700.366,E2 -14700.366} C_VEL
LIN {X 0,Y 333.641,Z 212.924,A -85,B 0,C 180,E1 -14703.208,E2 -14703.208} C_VEL
LIN {X 0,Y 333.683,Z 212.916,A -85,B 0,C 180,E1 -14704.829,E2 -14704.829} C_VEL
LIN {X 0,Y 332.965,Z 213.01,A -85,B 0,C 180,E1 -14705.836,E2 -14705.836} C_VEL
LIN {X 0,Y 330.073,Z 213.371,A -85,B 0,C 180,E1 -14707.473,E2 -14707.473} C_VEL
LIN {X 0,Y 327.665,Z 213.668,A -85,B 0,C 180,E1 -14708.799,E2 -14708.799} C_VEL
LIN {X 0,Y 326.656,Z 213.795,A -85,B 0,C 180,E1 -14709.826,E2 -14709.826} C_VEL
LIN {X 0,Y 326.585,Z 213.802,A -85,B 0,C 180,E1 -14710.174,E2 -14710.174} C_VEL
LIN {X 0,Y 326.563,Z 213.809,A -85,B 0,C 180,E1 -14713.526,E2 -14713.526} C_VEL
LIN {X 0,Y 326.576,Z 213.805,A -85,B 0,C 180,E1 -14717.029,E2 -14717.029} C_VEL
LIN {X 0,Y 326.584,Z 213.806,A -85,B 0,C 180,E1 -14721.386,E2 -14721.386} C_VEL
LIN {X 0,Y 326.621,Z 213.799,A -85,B 0,C 180,E1 -14724.852,E2 -14724.852} C_VEL
LIN {X 0,Y 326.61,Z 213.801,A -85,B 0,C 180,E1 -14727.456,E2 -14727.456} C_VEL
LIN {X 0,Y 326.619,Z 213.797,A -85,B 0,C 180,E1 -14730.337,E2 -14730.337} C_VEL
LIN {X 0,Y 326.644,Z 213.796,A -85,B 0,C 180,E1 -14734.645,E2 -14734.645} C_VEL
LIN {X 0,Y 326.622,Z 213.799,A -85,B 0,C 180,E1 -14738.544,E2 -14738.544} C_VEL
LIN {X 0,Y 326.71,Z 213.788,A -85,B 0,C 180,E1 -14741.175,E2 -14741.175} C_VEL
LIN {X 0,Y 326.766,Z 213.779,A -85,B 0,C 180,E1 -14745.433,E2 -14745.433} C_VEL
LIN {X 0,Y 326.761,Z 213.783,A -85,B 0,C 180,E1 -14748.839,E2 -14748.839} C_VEL
LIN {X 0,Y 326.917,Z 213.765,A -85,B 0,C 180,E1 -14752.589,E2 -14752.589} C_VEL
LIN {X 0,Y 326.761,Z 213.78,A -85,B 0,C 180,E1 -14755.065,E2 -14755.065} C_VEL
LIN {X 0,Y 327.037,Z 213.745,A -85,B 0,C 180,E1 -14757.537,E2 -14757.537} C_VEL
LIN {X 0,Y 327.047,Z 213.744,A -85,B 0,C 180,E1 -14761.231,E2 -14761.231} C_VEL
LIN {X 0,Y 326.756,Z 213.781,A -85,B 0,C 180,E1 -14763.7,E2 -14763.7} C_VEL
LIN {X 0,Y 326.946,Z 213.761,A -85,B 0,C 180,E1 -14766.17,E2 -14766.17} C_VEL
LIN {X 0,Y 326.807,Z 213.777,A -85,B 0,C 180,E1 -14769.907,E2 -14769.907} C_VEL
LIN {X 0,Y 326.746,Z 213.783,A -85,B 0,C 180,E1 -14773.686,E2 -14773.686} C_VEL
LIN {X 0,Y 326.654,Z 213.794,A -85,B 0,C 180,E1 -14777.531,E2 -14777.531} C_VEL
LIN {X 0,Y 326.631,Z 213.799,A -85,B 0,C 180,E1 -14780.137,E2 -14780.137} C_VEL
LIN {X 0,Y 326.613,Z 213.8,A -85,B 0,C 180,E1 -14784.132,E2 -14784.132} C_VEL
LIN {X 0,Y 326.601,Z 213.8,A -85,B 0,C 180,E1 -14788.256,E2 -14788.256} C_VEL
LIN {X 0,Y 326.576,Z 213.804,A -85,B 0,C 180,E1 -14791.097,E2 -14791.097} C_VEL
LIN {X 0,Y 326.61,Z 213.8,A -85,B 0,C 180,E1 -14794.019,E2 -14794.019} C_VEL
LIN {X 0,Y 326.625,Z 213.799,A -85,B 0,C 180,E1 -14797.237,E2 -14797.237} C_VEL
LIN {X 0,Y 326.546,Z 213.809,A -85,B 0,C 180,E1 -14801.124,E2 -14801.124} C_VEL
LIN {X 0,Y 326.561,Z 213.808,A -85,B 0,C 180,E1 -14803.526,E2 -14803.526} C_VEL
LIN {X 0,Y 326.575,Z 213.806,A -85,B 0,C 180,E1 -14807.029,E2 -14807.029} C_VEL
LIN {X 0,Y 326.584,Z 213.805,A -85,B 0,C 180,E1 -14811.385,E2 -14811.385} C_VEL
LIN {X 0,Y 326.62,Z 213.8,A -85,B 0,C 180,E1 -14814.852,E2 -14814.852} C_VEL
LIN {X 0,Y 326.673,Z 213.906,A -85,B 0,C 180,E1 -14816.944,E2 -14816.944} C_VEL
LIN {X 0,Y 329.791,Z 228.54,A -85,B 0,C 180,E1 -14820.65,E2 -14820.65} C_VEL
LIN {X 0,Y 331.14,Z 235.89,A -85,B 0,C 180,E1 -14822.439,E2 -14822.439} C_VEL
LIN {X 0,Y 330.477,Z 243.515,A -85,B 0,C 180,E1 -14824.153,E2 -14824.153} C_VEL
LIN {X 0,Y 329.309,Z 254.486,A -85,B 0,C 180,E1 -14826.591,E2 -14826.591} C_VEL
LIN {X 0,Y 334.568,Z 299.245,A -85,B 0,C 180,E1 -14828.047,E2 -14828.047} C_VEL
LIN {X 0,Y 333.021,Z 364.73,A -85,B 0,C 180,E1 -14829.662,E2 -14829.662} C_VEL
LIN {X 0,Y 332.17,Z 378.587,A -85,B 0,C 180,E1 -14830.253,E2 -14830.253} C_VEL
LIN {X 0,Y 331.354,Z 390.072,A -85,B 0,C 180,E1 -14830.967,E2 -14830.967} C_VEL
LIN {X 0,Y 330.257,Z 401.106,A -85,B 0,C 180,E1 -14831.867,E2 -14831.867} C_VEL
LIN {X 0,Y 329.09,Z 412.713,A -85,B 0,C 180,E1 -14833.083,E2 -14833.083} C_VEL
LIN {X 0,Y 327.935,Z 423.209,A -85,B 0,C 180,E1 -14834.462,E2 -14834.462} C_VEL
LIN {X 0,Y 327.093,Z 432.664,A -85,B 0,C 180,E1 -14836.012,E2 -14836.012} C_VEL
LIN {X 0,Y 326.329,Z 440.426,A -85,B 0,C 180,E1 -14837.563,E2 -14837.563} C_VEL
LIN {X 0,Y 325.598,Z 448.011,A -85,B 0,C 180,E1 -14839.428,E2 -14839.428} C_VEL
LIN {X 0,Y 325.285,Z 454.098,A -85,B 0,C 180,E1 -14841.301,E2 -14841.301} C_VEL
LIN {X 0,Y 325.163,Z 458.869,A -85,B 0,C 180,E1 -14843.172,E2 -14843.172} C_VEL
LIN {X 0,Y 325.198,Z 462.465,A -85,B 0,C 180,E1 -14845.04,E2 -14845.04} C_VEL
LIN {X 0,Y 325.133,Z 464.247,A -85,B 0,C 180,E1 -14846.282,E2 -14846.282} C_VEL
LIN {X 0,Y 325.3,Z 465.584,A -85,B 0,C 180,E1 -14847.523,E2 -14847.523} C_VEL
LIN {X 0,Y 325.329,Z 466.486,A -85,B 0,C 180,E1 -14848.762,E2 -14848.762} C_VEL
LIN {X 0,Y 325.331,Z 466.968,A -85,B 0,C 180,E1 -14850,E2 -14850} C_VEL
LIN {X 0,Y 325.305,Z 466.985,A -85,B 0,C 180,E1 -14851.238,E2 -14851.238} C_VEL
LIN {X 0,Y 325.186,Z 466.58,A -85,B 0,C 180,E1 -14852.477,E2 -14852.477} C_VEL
LIN {X 0,Y 325.076,Z 465.771,A -85,B 0,C 180,E1 -14853.718,E2 -14853.718} C_VEL
LIN {X 0,Y 324.99,Z 463.38,A -85,B 0,C 180,E1 -14855.864,E2 -14855.864} C_VEL
LIN {X 0,Y 325.184,Z 459.521,A -85,B 0,C 180,E1 -14858.075,E2 -14858.075} C_VEL
LIN {X 0,Y 325.487,Z 455.095,A -85,B 0,C 180,E1 -14859.947,E2 -14859.947} C_VEL
LIN {X 0,Y 326.303,Z 448.419,A -85,B 0,C 180,E1 -14862.122,E2 -14862.122} C_VEL
LIN {X 0,Y 327.351,Z 441.215,A -85,B 0,C 180,E1 -14863.977,E2 -14863.977} C_VEL
LIN {X 0,Y 328.476,Z 433.104,A -85,B 0,C 180,E1 -14865.674,E2 -14865.674} C_VEL
LIN {X 0,Y 330.035,Z 423.199,A -85,B 0,C 180,E1 -14867.345,E2 -14867.345} C_VEL
LIN {X 0,Y 331.824,Z 412.078,A -85,B 0,C 180,E1 -14868.844,E2 -14868.844} C_VEL
LIN {X 0,Y 333.397,Z 400.933,A -85,B 0,C 180,E1 -14870.032,E2 -14870.032} C_VEL
LIN {X 0,Y 334.991,Z 388.6,A -85,B 0,C 180,E1 -14871.055,E2 -14871.055} C_VEL
LIN {X 0,Y 336.41,Z 375.709,A -85,B 0,C 180,E1 -14871.846,E2 -14871.846} C_VEL
LIN {X 0,Y 337.448,Z 362.146,A -85,B 0,C 180,E1 -14872.42,E2 -14872.42} C_VEL
LIN {X 0,Y 339.504,Z 298.848,A -85,B 0,C 180,E1 -14874.043,E2 -14874.043} C_VEL
LIN {X 0,Y 337.285,Z 279.385,A -85,B 0,C 180,E1 -14874.821,E2 -14874.821} C_VEL
LIN {X 0,Y 333.982,Z 259.86,A -85,B 0,C 180,E1 -14875.731,E2 -14875.731} C_VEL
LIN {X 0,Y 331.923,Z 249.51,A -85,B 0,C 180,E1 -14876.288,E2 -14876.288} C_VEL
LIN {X 0,Y 332.929,Z 240.2,A -85,B 0,C 180,E1 -14878.357,E2 -14878.357} C_VEL
LIN {X 0,Y 330.922,Z 230.115,A -85,B 0,C 180,E1 -14880.976,E2 -14880.976} C_VEL
LIN {X 0,Y 328.382,Z 219.999,A -85,B 0,C 180,E1 -14883.81,E2 -14883.81} C_VEL
LIN {X 0,Y 326.632,Z 213.797,A -85,B 0,C 180,E1 -14885.706,E2 -14885.706} C_VEL
LIN {X 0,Y 326.571,Z 213.803,A -85,B 0,C 180,E1 -14889.218,E2 -14889.218} C_VEL
LIN {X 0,Y 326.574,Z 213.801,A -85,B 0,C 180,E1 -14892.971,E2 -14892.971} C_VEL
LIN {X 0,Y 326.573,Z 213.801,A -85,B 0,C 180,E1 -14897.028,E2 -14897.028} C_VEL
LIN {X 0,Y 326.582,Z 213.804,A -85,B 0,C 180,E1 -14901.385,E2 -14901.385} C_VEL
LIN {X 0,Y 326.619,Z 213.796,A -85,B 0,C 180,E1 -14904.851,E2 -14904.851} C_VEL
LIN {X 0,Y 326.609,Z 213.797,A -85,B 0,C 180,E1 -14907.456,E2 -14907.456} C_VEL
LIN {X 0,Y 326.617,Z 213.795,A -85,B 0,C 180,E1 -14910.336,E2 -14910.336} C_VEL
LIN {X 0,Y 326.617,Z 213.795,A -85,B 0,C 180,E1 -14913.136,E2 -14913.136} C_VEL
LIN {X 0,Y 326.639,Z 213.794,A -85,B 0,C 180,E1 -14915.87,E2 -14915.87} C_VEL
LIN {X 0,Y 326.649,Z 213.792,A -85,B 0,C 180,E1 -14919.864,E2 -14919.864} C_VEL
LIN {X 0,Y 326.663,Z 213.788,A -85,B 0,C 180,E1 -14922.47,E2 -14922.47} C_VEL
LIN {X 0,Y 326.759,Z 213.781,A -85,B 0,C 180,E1 -14926.314,E2 -14926.314} C_VEL
LIN {X 0,Y 326.806,Z 213.775,A -85,B 0,C 180,E1 -14930.093,E2 -14930.093} C_VEL
LIN {X 0,Y 326.988,Z 213.751,A -85,B 0,C 180,E1 -14933.831,E2 -14933.831} C_VEL
LIN {X 0,Y 327.045,Z 213.749,A -85,B 0,C 180,E1 -14937.537,E2 -14937.537} C_VEL
LIN {X 0,Y 327.197,Z 213.729,A -85,B 0,C 180,E1 -14940,E2 -14940} C_VEL
LIN {X 0,Y 327.045,Z 213.747,A -85,B 0,C 180,E1 -14942.463,E2 -14942.463} C_VEL
LIN {X 0,Y 326.937,Z 213.758,A -85,B 0,C 180,E1 -14946.482,E2 -14946.482} C_VEL
LIN {X 0,Y 326.783,Z 213.783,A -85,B 0,C 180,E1 -14949.907,E2 -14949.907} C_VEL
LIN {X 0,Y 326.769,Z 213.787,A -85,B 0,C 180,E1 -14951.239,E2 -14951.239} C_VEL
LIN {X 0,Y 327.782,Z 216.665,A -85,B 0,C 180,E1 -14951.459,E2 -14951.459} C_VEL
LIN {X 0,Y 329.394,Z 219.323,A -85,B 0,C 180,E1 -14951.732,E2 -14951.732} C_VEL
LIN {X 0,Y 336.926,Z 233.305,A -85,B 0,C 180,E1 -14953.009,E2 -14953.009} C_VEL
LIN {X 0,Y 341.277,Z 242.901,A -85,B 0,C 180,E1 -14953.737,E2 -14953.737} C_VEL
LIN {X 0,Y 338.536,Z 319.22,A -85,B 0,C 180,E1 -14955.687,E2 -14955.687} C_VEL
LIN {X 0,Y 337.913,Z 332.452,A -85,B 0,C 180,E1 -14956.279,E2 -14956.279} C_VEL
LIN {X 0,Y 336.997,Z 344.661,A -85,B 0,C 180,E1 -14957.054,E2 -14957.054} C_VEL
LIN {X 0,Y 335.857,Z 355.727,A -85,B 0,C 180,E1 -14957.978,E2 -14957.978} C_VEL
LIN {X 0,Y 334.63,Z 366.068,A -85,B 0,C 180,E1 -14959.074,E2 -14959.074} C_VEL
LIN {X 0,Y 333.081,Z 377.114,A -85,B 0,C 180,E1 -14960.535,E2 -14960.535} C_VEL
LIN {X 0,Y 331.614,Z 386.771,A -85,B 0,C 180,E1 -14962.155,E2 -14962.155} C_VEL
LIN {X 0,Y 330.222,Z 394.931,A -85,B 0,C 180,E1 -14963.852,E2 -14963.852} C_VEL
LIN {X 0,Y 328.924,Z 402.045,A -85,B 0,C 180,E1 -14965.689,E2 -14965.689} C_VEL
LIN {X 0,Y 327.948,Z 407.418,A -85,B 0,C 180,E1 -14967.435,E2 -14967.435} C_VEL
LIN {X 0,Y 326.951,Z 412.597,A -85,B 0,C 180,E1 -14969.63,E2 -14969.63} C_VEL
LIN {X 0,Y 326.172,Z 416.32,A -85,B 0,C 180,E1 -14971.864,E2 -14971.864} C_VEL
LIN {X 0,Y 325.585,Z 418.664,A -85,B 0,C 180,E1 -14974.141,E2 -14974.141} C_VEL
LIN {X 0,Y 325.356,Z 419.406,A -85,B 0,C 180,E1 -14975.678,E2 -14975.678} C_VEL
LIN {X 0,Y 325.19,Z 419.557,A -85,B 0,C 180,E1 -14977.239,E2 -14977.239} C_VEL
LIN {X 0,Y 325.147,Z 418.988,A -85,B 0,C 180,E1 -14978.91,E2 -14978.91} C_VEL
LIN {X 0,Y 325.221,Z 417.382,A -85,B 0,C 180,E1 -14980.857,E2 -14980.857} C_VEL
LIN {X 0,Y 325.536,Z 414.769,A -85,B 0,C 180,E1 -14982.775,E2 -14982.775} C_VEL
LIN {X 0,Y 325.88,Z 411.22,A -85,B 0,C 180,E1 -14984.628,E2 -14984.628} C_VEL
LIN {X 0,Y 326.334,Z 406.684,A -85,B 0,C 180,E1 -14986.437,E2 -14986.437} C_VEL
LIN {X 0,Y 327.015,Z 399.906,A -85,B 0,C 180,E1 -14988.532,E2 -14988.532} C_VEL
LIN {X 0,Y 327.902,Z 391.803,A -85,B 0,C 180,E1 -14990.498,E2 -14990.498} C_VEL
LIN {X 0,Y 328.865,Z 382.721,A -85,B 0,C 180,E1 -14992.252,E2 -14992.252} C_VEL
LIN {X 0,Y 329.998,Z 371.92,A -85,B 0,C 180,E1 -14993.916,E2 -14993.916} C_VEL
LIN {X 0,Y 330.924,Z 361.413,A -85,B 0,C 180,E1 -14995.216,E2 -14995.216} C_VEL
LIN {X 0,Y 331.921,Z 349.584,A -85,B 0,C 180,E1 -14996.367,E2 -14996.367} C_VEL
LIN {X 0,Y 332.73,Z 337.085,A -85,B 0,C 180,E1 -14997.307,E2 -14997.307} C_VEL
LIN {X 0,Y 333.249,Z 324.402,A -85,B 0,C 180,E1 -14998,E2 -14998} C_VEL
LIN {X 0,Y 333.688,Z 310.318,A -85,B 0,C 180,E1 -14998.494,E2 -14998.494} C_VEL
LIN {X 0,Y 335.522,Z 237.289,A -85,B 0,C 180,E1 -15000.253,E2 -15000.253} C_VEL
LIN {X 0,Y 326.689,Z 213.792,A -85,B 0,C 180,E1 -15001.403,E2 -15001.403} C_VEL
LIN {X 0,Y 326.688,Z 213.79,A -85,B 0,C 180,E1 -15004.628,E2 -15004.628} C_VEL
LIN {X 0,Y 326.62,Z 213.798,A -85,B 0,C 180,E1 -15008.544,E2 -15008.544} C_VEL
LIN {X 0,Y 326.707,Z 213.789,A -85,B 0,C 180,E1 -15011.176,E2 -15011.176} C_VEL
LIN {X 0,Y 326.764,Z 213.78,A -85,B 0,C 180,E1 -15015.434,E2 -15015.434} C_VEL
LIN {X 0,Y 326.759,Z 213.784,A -85,B 0,C 180,E1 -15018.839,E2 -15018.839} C_VEL
LIN {X 0,Y 326.919,Z 213.764,A -85,B 0,C 180,E1 -15022.589,E2 -15022.589} C_VEL
LIN {X 0,Y 326.765,Z 213.78,A -85,B 0,C 180,E1 -15025.065,E2 -15025.065} C_VEL
LIN {X 0,Y 327.043,Z 213.744,A -85,B 0,C 180,E1 -15027.537,E2 -15027.537} C_VEL
LIN {X 0,Y 327.16,Z 213.731,A -85,B 0,C 180,E1 -15030,E2 -15030} C_VEL
LIN {X 0,Y 327.034,Z 213.751,A -85,B 0,C 180,E1 -15032.464,E2 -15032.464} C_VEL
LIN {X 0,Y 326.953,Z 213.759,A -85,B 0,C 180,E1 -15036.17,E2 -15036.17} C_VEL
LIN {X 0,Y 326.806,Z 213.776,A -85,B 0,C 180,E1 -15039.907,E2 -15039.907} C_VEL
LIN {X 0,Y 326.761,Z 213.781,A -85,B 0,C 180,E1 -15043.686,E2 -15043.686} C_VEL
LIN {X 0,Y 326.701,Z 213.788,A -85,B 0,C 180,E1 -15047.528,E2 -15047.528} C_VEL
LIN {X 0,Y 326.66,Z 213.796,A -85,B 0,C 180,E1 -15050.136,E2 -15050.136} C_VEL
LIN {X 0,Y 326.645,Z 213.797,A -85,B 0,C 180,E1 -15054.13,E2 -15054.13} C_VEL
LIN {X 0,Y 326.623,Z 213.798,A -85,B 0,C 180,E1 -15058.254,E2 -15058.254} C_VEL
LIN {X 0,Y 326.576,Z 213.803,A -85,B 0,C 180,E1 -15061.097,E2 -15061.097} C_VEL
LIN {X 0,Y 326.609,Z 213.801,A -85,B 0,C 180,E1 -15064.02,E2 -15064.02} C_VEL
LIN {X 0,Y 326.625,Z 213.798,A -85,B 0,C 180,E1 -15067.238,E2 -15067.238} C_VEL
LIN {X 0,Y 326.585,Z 213.802,A -85,B 0,C 180,E1 -15070.174,E2 -15070.174} C_VEL
LIN {X 0,Y 325.939,Z 213.886,A -85,B 0,C 180,E1 -15071.204,E2 -15071.204} C_VEL
LIN {X 0,Y 323.065,Z 214.248,A -85,B 0,C 180,E1 -15072.878,E2 -15072.878} C_VEL
LIN {X 0,Y 320.614,Z 214.552,A -85,B 0,C 180,E1 -15074.234,E2 -15074.234} C_VEL
LIN {X 0,Y 319.565,Z 214.68,A -85,B 0,C 180,E1 -15075.285,E2 -15075.285} C_VEL
LIN {X 0,Y 319.483,Z 214.686,A -85,B 0,C 180,E1 -15075.641,E2 -15075.641} C_VEL
LIN {X 0,Y 319.501,Z 214.684,A -85,B 0,C 180,E1 -15078.707,E2 -15078.707} C_VEL
LIN {X 0,Y 319.548,Z 214.677,A -85,B 0,C 180,E1 -15082.352,E2 -15082.352} C_VEL
LIN {X 0,Y 319.562,Z 214.681,A -85,B 0,C 180,E1 -15085.124,E2 -15085.124} C_VEL
LIN {X 0,Y 319.526,Z 214.68,A -85,B 0,C 180,E1 -15088.138,E2 -15088.138} C_VEL
LIN {X 0,Y 319.573,Z 214.675,A -85,B 0,C 180,E1 -15091.604,E2 -15091.604} C_VEL
LIN {X 0,Y 319.576,Z 214.676,A -85,B 0,C 180,E1 -15095.302,E2 -15095.302} C_VEL
LIN {X 0,Y 319.57,Z 214.675,A -85,B 0,C 180,E1 -15098.046,E2 -15098.046} C_VEL
LIN {X 0,Y 319.66,Z 214.668,A -85,B 0,C 180,E1 -15100.979,E2 -15100.979} C_VEL
LIN {X 0,Y 319.715,Z 214.658,A -85,B 0,C 180,E1 -15105.289,E2 -15105.289} C_VEL
LIN {X 0,Y 319.718,Z 214.661,A -85,B 0,C 180,E1 -15108.59,E2 -15108.59} C_VEL
LIN {X 0,Y 319.856,Z 214.643,A -85,B 0,C 180,E1 -15112.424,E2 -15112.424} C_VEL
LIN {X 0,Y 319.73,Z 214.656,A -85,B 0,C 180,E1 -15114.956,E2 -15114.956} C_VEL
LIN {X 0,Y 319.981,Z 214.624,A -85,B 0,C 180,E1 -15117.482,E2 -15117.482} C_VEL
LIN {X 0,Y 320.014,Z 214.62,A -85,B 0,C 180,E1 -15121.258,E2 -15121.258} C_VEL
LIN {X 0,Y 319.722,Z 214.656,A -85,B 0,C 180,E1 -15125.044,E2 -15125.044} C_VEL
LIN {X 0,Y 319.856,Z 214.64,A -85,B 0,C 180,E1 -15127.576,E2 -15127.576} C_VEL
LIN {X 0,Y 319.725,Z 214.656,A -85,B 0,C 180,E1 -15131.41,E2 -15131.41} C_VEL
LIN {X 0,Y 319.668,Z 214.663,A -85,B 0,C 180,E1 -15134.679,E2 -15134.679} C_VEL
LIN {X 0,Y 319.619,Z 214.675,A -85,B 0,C 180,E1 -15137.929,E2 -15137.929} C_VEL
LIN {X 0,Y 319.586,Z 214.673,A -85,B 0,C 180,E1 -15140.601,E2 -15140.601} C_VEL
LIN {X 0,Y 319.543,Z 214.68,A -85,B 0,C 180,E1 -15143.322,E2 -15143.322} C_VEL
LIN {X 0,Y 319.555,Z 214.679,A -85,B 0,C 180,E1 -15146.095,E2 -15146.095} C_VEL
LIN {X 0,Y 319.545,Z 214.678,A -85,B 0,C 180,E1 -15148.938,E2 -15148.938} C_VEL
LIN {X 0,Y 319.526,Z 214.684,A -85,B 0,C 180,E1 -15151.863,E2 -15151.863} C_VEL
LIN {X 0,Y 319.582,Z 214.679,A -85,B 0,C 180,E1 -15155.543,E2 -15155.543} C_VEL
LIN {X 0,Y 319.53,Z 214.683,A -85,B 0,C 180,E1 -15159.662,E2 -15159.662} C_VEL
LIN {X 0,Y 319.521,Z 214.686,A -85,B 0,C 180,E1 -15163.46,E2 -15163.46} C_VEL
LIN {X 0,Y 319.553,Z 214.68,A -85,B 0,C 180,E1 -15167.016,E2 -15167.016} C_VEL
LIN {X 0,Y 319.547,Z 214.678,A -85,B 0,C 180,E1 -15170.37,E2 -15170.37} C_VEL
LIN {X 0,Y 319.58,Z 214.675,A -85,B 0,C 180,E1 -15174.457,E2 -15174.457} C_VEL
LIN {X 0,Y 319.612,Z 214.748,A -85,B 0,C 180,E1 -15176.604,E2 -15176.604} C_VEL
LIN {X 0,Y 322.37,Z 227.434,A -85,B 0,C 180,E1 -15179.905,E2 -15179.905} C_VEL
LIN {X 0,Y 324.137,Z 236.643,A -85,B 0,C 180,E1 -15182.209,E2 -15182.209} C_VEL
LIN {X 0,Y 323.896,Z 241.087,A -85,B 0,C 180,E1 -15183.241,E2 -15183.241} C_VEL
LIN {X 0,Y 322.452,Z 254.243,A -85,B 0,C 180,E1 -15186.184,E2 -15186.184} C_VEL
LIN {X 0,Y 327.774,Z 299.086,A -85,B 0,C 180,E1 -15187.685,E2 -15187.685} C_VEL
LIN {X 0,Y 326.177,Z 364.377,A -85,B 0,C 180,E1 -15189.339,E2 -15189.339} C_VEL
LIN {X 0,Y 325.307,Z 378.157,A -85,B 0,C 180,E1 -15189.942,E2 -15189.942} C_VEL
LIN {X 0,Y 324.427,Z 390.126,A -85,B 0,C 180,E1 -15190.709,E2 -15190.709} C_VEL
LIN {X 0,Y 323.212,Z 402.628,A -85,B 0,C 180,E1 -15191.785,E2 -15191.785} C_VEL
LIN {X 0,Y 321.911,Z 413.848,A -85,B 0,C 180,E1 -15193.022,E2 -15193.022} C_VEL
LIN {X 0,Y 320.813,Z 424.002,A -85,B 0,C 180,E1 -15194.434,E2 -15194.434} C_VEL
LIN {X 0,Y 319.955,Z 433.215,A -85,B 0,C 180,E1 -15196.017,E2 -15196.017} C_VEL
LIN {X 0,Y 319.077,Z 442.189,A -85,B 0,C 180,E1 -15197.921,E2 -15197.921} C_VEL
LIN {X 0,Y 318.441,Z 449.318,A -85,B 0,C 180,E1 -15199.83,E2 -15199.83} C_VEL
LIN {X 0,Y 318.154,Z 455.005,A -85,B 0,C 180,E1 -15201.744,E2 -15201.744} C_VEL
LIN {X 0,Y 318.105,Z 459.777,A -85,B 0,C 180,E1 -15203.829,E2 -15203.829} C_VEL
LIN {X 0,Y 318.104,Z 461.755,A -85,B 0,C 180,E1 -15204.93,E2 -15204.93} C_VEL
LIN {X 0,Y 318.059,Z 463.595,A -85,B 0,C 180,E1 -15206.199,E2 -15206.199} C_VEL
LIN {X 0,Y 318.205,Z 464.958,A -85,B 0,C 180,E1 -15207.468,E2 -15207.468} C_VEL
LIN {X 0,Y 318.268,Z 465.89,A -85,B 0,C 180,E1 -15208.734,E2 -15208.734} C_VEL
LIN {X 0,Y 318.268,Z 466.401,A -85,B 0,C 180,E1 -15210,E2 -15210} C_VEL
LIN {X 0,Y 318.241,Z 466.465,A -85,B 0,C 180,E1 -15211.265,E2 -15211.265} C_VEL
LIN {X 0,Y 318.09,Z 466.082,A -85,B 0,C 180,E1 -15212.532,E2 -15212.532} C_VEL
LIN {X 0,Y 317.995,Z 465.296,A -85,B 0,C 180,E1 -15213.801,E2 -15213.801} C_VEL
LIN {X 0,Y 317.903,Z 463.169,A -85,B 0,C 180,E1 -15215.825,E2 -15215.825} C_VEL
LIN {X 0,Y 318.029,Z 460.361,A -85,B 0,C 180,E1 -15217.619,E2 -15217.619} C_VEL
LIN {X 0,Y 318.297,Z 456.353,A -85,B 0,C 180,E1 -15219.532,E2 -15219.532} C_VEL
LIN {X 0,Y 318.832,Z 451.228,A -85,B 0,C 180,E1 -15221.442,E2 -15221.442} C_VEL
LIN {X 0,Y 319.885,Z 444.834,A -85,B 0,C 180,E1 -15223.337,E2 -15223.337} C_VEL
LIN {X 0,Y 321.104,Z 436.938,A -85,B 0,C 180,E1 -15225.227,E2 -15225.227} C_VEL
LIN {X 0,Y 322.337,Z 428.915,A -85,B 0,C 180,E1 -15226.791,E2 -15226.791} C_VEL
LIN {X 0,Y 324.154,Z 418.096,A -85,B 0,C 180,E1 -15228.486,E2 -15228.486} C_VEL
LIN {X 0,Y 325.907,Z 407.172,A -85,B 0,C 180,E1 -15229.855,E2 -15229.855} C_VEL
LIN {X 0,Y 327.71,Z 394.896,A -85,B 0,C 180,E1 -15231.052,E2 -15231.052} C_VEL
LIN {X 0,Y 329.375,Z 382.022,A -85,B 0,C 180,E1 -15232.008,E2 -15232.008} C_VEL
LIN {X 0,Y 330.703,Z 369.044,A -85,B 0,C 180,E1 -15232.696,E2 -15232.696} C_VEL
LIN {X 0,Y 331.474,Z 355.676,A -85,B 0,C 180,E1 -15233.176,E2 -15233.176} C_VEL
LIN {X 0,Y 333.288,Z 299.519,A -85,B 0,C 180,E1 -15234.627,E2 -15234.627} C_VEL
LIN {X 0,Y 330.898,Z 278.479,A -85,B 0,C 180,E1 -15235.498,E2 -15235.498} C_VEL
LIN {X 0,Y 327.233,Z 257.566,A -85,B 0,C 180,E1 -15236.544,E2 -15236.544} C_VEL
LIN {X 0,Y 325.427,Z 248.789,A -85,B 0,C 180,E1 -15237.055,E2 -15237.055} C_VEL
LIN {X 0,Y 326.181,Z 243.275,A -85,B 0,C 180,E1 -15238.295,E2 -15238.295} C_VEL
LIN {X 0,Y 325.39,Z 237.479,A -85,B 0,C 180,E1 -15239.786,E2 -15239.786} C_VEL
LIN {X 0,Y 322.765,Z 226.014,A -85,B 0,C 180,E1 -15242.98,E2 -15242.98} C_VEL
LIN {X 0,Y 319.607,Z 214.675,A -85,B 0,C 180,E1 -15246.47,E2 -15246.47} C_VEL
LIN {X 0,Y 319.528,Z 214.682,A -85,B 0,C 180,E1 -15249.662,E2 -15249.662} C_VEL
LIN {X 0,Y 319.52,Z 214.681,A -85,B 0,C 180,E1 -15253.46,E2 -15253.46} C_VEL
LIN {X 0,Y 319.552,Z 214.675,A -85,B 0,C 180,E1 -15257.016,E2 -15257.016} C_VEL
LIN {X 0,Y 319.544,Z 214.678,A -85,B 0,C 180,E1 -15260.37,E2 -15260.37} C_VEL
LIN {X 0,Y 319.579,Z 214.674,A -85,B 0,C 180,E1 -15264.457,E2 -15264.457} C_VEL
LIN {X 0,Y 319.525,Z 214.68,A -85,B 0,C 180,E1 -15268.137,E2 -15268.137} C_VEL
LIN {X 0,Y 319.588,Z 214.674,A -85,B 0,C 180,E1 -15271.597,E2 -15271.597} C_VEL
LIN {X 0,Y 319.58,Z 214.677,A -85,B 0,C 180,E1 -15275.302,E2 -15275.302} C_VEL
LIN {X 0,Y 319.597,Z 214.67,A -85,B 0,C 180,E1 -15279.4,E2 -15279.4} C_VEL
LIN {X 0,Y 319.624,Z 214.666,A -85,B 0,C 180,E1 -15282.071,E2 -15282.071} C_VEL
LIN {X 0,Y 319.732,Z 214.654,A -85,B 0,C 180,E1 -15286.008,E2 -15286.008} C_VEL
LIN {X 0,Y 319.752,Z 214.655,A -85,B 0,C 180,E1 -15289.873,E2 -15289.873} C_VEL
LIN {X 0,Y 319.912,Z 214.635,A -85,B 0,C 180,E1 -15292.426,E2 -15292.426} C_VEL
LIN {X 0,Y 319.744,Z 214.657,A -85,B 0,C 180,E1 -15294.956,E2 -15294.956} C_VEL
LIN {X 0,Y 319.988,Z 214.629,A -85,B 0,C 180,E1 -15297.482,E2 -15297.482} C_VEL
LIN {X 0,Y 320.149,Z 214.607,A -85,B 0,C 180,E1 -15300,E2 -15300} C_VEL
LIN {X 0,Y 319.989,Z 214.626,A -85,B 0,C 180,E1 -15302.518,E2 -15302.518} C_VEL
LIN {X 0,Y 319.902,Z 214.635,A -85,B 0,C 180,E1 -15306.468,E2 -15306.468} C_VEL
LIN {X 0,Y 319.74,Z 214.66,A -85,B 0,C 180,E1 -15310.367,E2 -15310.367} C_VEL
LIN {X 0,Y 320.761,Z 217.591,A -85,B 0,C 180,E1 -15310.613,E2 -15310.613} C_VEL
LIN {X 0,Y 322.316,Z 220.019,A -85,B 0,C 180,E1 -15310.893,E2 -15310.893} C_VEL
LIN {X 0,Y 329.349,Z 232.678,A -85,B 0,C 180,E1 -15312.145,E2 -15312.145} C_VEL
LIN {X 0,Y 335.053,Z 244.577,A -85,B 0,C 180,E1 -15313.147,E2 -15313.147} C_VEL
LIN {X 0,Y 332.3,Z 319.724,A -85,B 0,C 180,E1 -15315.114,E2 -15315.114} C_VEL
LIN {X 0,Y 331.659,Z 332.909,A -85,B 0,C 180,E1 -15315.714,E2 -15315.714} C_VEL
LIN {X 0,Y 330.691,Z 345.175,A -85,B 0,C 180,E1 -15316.504,E2 -15316.504} C_VEL
LIN {X 0,Y 329.355,Z 357.219,A -85,B 0,C 180,E1 -15317.542,E2 -15317.542} C_VEL
LIN {X 0,Y 327.98,Z 368.093,A -85,B 0,C 180,E1 -15318.749,E2 -15318.749} C_VEL
LIN {X 0,Y 326.455,Z 378.235,A -85,B 0,C 180,E1 -15320.148,E2 -15320.148} C_VEL
LIN {X 0,Y 325.075,Z 386.852,A -85,B 0,C 180,E1 -15321.621,E2 -15321.621} C_VEL
LIN {X 0,Y 323.461,Z 395.701,A -85,B 0,C 180,E1 -15323.49,E2 -15323.49} C_VEL
LIN {X 0,Y 322.007,Z 403.341,A -85,B 0,C 180,E1 -15325.535,E2 -15325.535} C_VEL
LIN {X 0,Y 320.952,Z 408.716,A -85,B 0,C 180,E1 -15327.377,E2 -15327.377} C_VEL
LIN {X 0,Y 319.924,Z 413.695,A -85,B 0,C 180,E1 -15329.622,E2 -15329.622} C_VEL
LIN {X 0,Y 319.105,Z 417.256,A -85,B 0,C 180,E1 -15331.909,E2 -15331.909} C_VEL
LIN {X 0,Y 318.667,Z 418.815,A -85,B 0,C 180,E1 -15333.46,E2 -15333.46} C_VEL
LIN {X 0,Y 318.34,Z 419.859,A -85,B 0,C 180,E1 -15335.23,E2 -15335.23} C_VEL
LIN {X 0,Y 318.126,Z 420.057,A -85,B 0,C 180,E1 -15337.316,E2 -15337.316} C_VEL
LIN {X 0,Y 318.086,Z 418.829,A -85,B 0,C 180,E1 -15339.847,E2 -15339.847} C_VEL
LIN {X 0,Y 318.382,Z 415.984,A -85,B 0,C 180,E1 -15342.319,E2 -15342.319} C_VEL
LIN {X 0,Y 318.68,Z 413.087,A -85,B 0,C 180,E1 -15344.015,E2 -15344.015} C_VEL
LIN {X 0,Y 319.194,Z 408.04,A -85,B 0,C 180,E1 -15346.2,E2 -15346.2} C_VEL
LIN {X 0,Y 319.848,Z 401.563,A -85,B 0,C 180,E1 -15348.338,E2 -15348.338} C_VEL
LIN {X 0,Y 320.584,Z 394.755,A -85,B 0,C 180,E1 -15350.111,E2 -15350.111} C_VEL
LIN {X 0,Y 321.562,Z 386.3,A -85,B 0,C 180,E1 -15351.888,E2 -15351.888} C_VEL
LIN {X 0,Y 322.527,Z 377.452,A -85,B 0,C 180,E1 -15353.409,E2 -15353.409} C_VEL
LIN {X 0,Y 323.48,Z 367.539,A -85,B 0,C 180,E1 -15354.806,E2 -15354.806} C_VEL
LIN {X 0,Y 324.574,Z 355.864,A -85,B 0,C 180,E1 -15356.113,E2 -15356.113} C_VEL
LIN {X 0,Y 325.499,Z 343.826,A -85,B 0,C 180,E1 -15357.166,E2 -15357.166} C_VEL
LIN {X 0,Y 326.218,Z 331.877,A -85,B 0,C 180,E1 -15357.96,E2 -15357.96} C_VEL
LIN {X 0,Y 326.684,Z 319.214,A -85,B 0,C 180,E1 -15358.554,E2 -15358.554} C_VEL
LIN {X 0,Y 327.111,Z 302.118,A -85,B 0,C 180,E1 -15359.038,E2 -15359.038} C_VEL
LIN {X 0,Y 328.643,Z 238.665,A -85,B 0,C 180,E1 -15360.611,E2 -15360.611} C_VEL
LIN {X 0,Y 319.635,Z 214.668,A -85,B 0,C 180,E1 -15361.828,E2 -15361.828} C_VEL
LIN {X 0,Y 319.603,Z 214.675,A -85,B 0,C 180,E1 -15365.304,E2 -15365.304} C_VEL
LIN {X 0,Y 319.589,Z 214.675,A -85,B 0,C 180,E1 -15369.4,E2 -15369.4} C_VEL
LIN {X 0,Y 319.625,Z 214.668,A -85,B 0,C 180,E1 -15372.071,E2 -15372.071} C_VEL
LIN {X 0,Y 319.733,Z 214.655,A -85,B 0,C 180,E1 -15376.008,E2 -15376.008} C_VEL
LIN {X 0,Y 319.736,Z 214.654,A -85,B 0,C 180,E1 -15379.872,E2 -15379.872} C_VEL
LIN {X 0,Y 319.908,Z 214.633,A -85,B 0,C 180,E1 -15383.694,E2 -15383.694} C_VEL
LIN {X 0,Y 319.987,Z 214.623,A -85,B 0,C 180,E1 -15387.483,E2 -15387.483} C_VEL
LIN {X 0,Y 320.113,Z 214.609,A -85,B 0,C 180,E1 -15390,E2 -15390} C_VEL
LIN {X 0,Y 319.977,Z 214.629,A -85,B 0,C 180,E1 -15392.518,E2 -15392.518} C_VEL
LIN {X 0,Y 319.909,Z 214.638,A -85,B 0,C 180,E1 -15396.307,E2 -15396.307} C_VEL
LIN {X 0,Y 319.753,Z 214.656,A -85,B 0,C 180,E1 -15400.128,E2 -15400.128} C_VEL
LIN {X 0,Y 319.733,Z 214.656,A -85,B 0,C 180,E1 -15404.725,E2 -15404.725} C_VEL
LIN {X 0,Y 319.69,Z 214.66,A -85,B 0,C 180,E1 -15409.038,E2 -15409.038} C_VEL
LIN {X 0,Y 319.559,Z 214.677,A -85,B 0,C 180,E1 -15413.321,E2 -15413.321} C_VEL
LIN {X 0,Y 319.577,Z 214.678,A -85,B 0,C 180,E1 -15416.094,E2 -15416.094} C_VEL
LIN {X 0,Y 319.554,Z 214.677,A -85,B 0,C 180,E1 -15418.938,E2 -15418.938} C_VEL
LIN {X 0,Y 319.527,Z 214.685,A -85,B 0,C 180,E1 -15421.863,E2 -15421.863} C_VEL
LIN {X 0,Y 319.581,Z 214.678,A -85,B 0,C 180,E1 -15425.543,E2 -15425.543} C_VEL
LIN {X 0,Y 319.56,Z 214.68,A -85,B 0,C 180,E1 -15429.669,E2 -15429.669} C_VEL
LIN {X 0,Y 319.523,Z 214.686,A -85,B 0,C 180,E1 -15433.461,E2 -15433.461} C_VEL
LIN {X 0,Y 319.483,Z 214.686,A -85,B 0,C 180,E1 -15435.641,E2 -15435.641} C_VEL
LIN {X 0,Y 318.831,Z 214.768,A -85,B 0,C 180,E1 -15436.694,E2 -15436.694} C_VEL
LIN {X 0,Y 316.015,Z 215.119,A -85,B 0,C 180,E1 -15438.408,E2 -15438.408} C_VEL
LIN {X 0,Y 313.615,Z 215.42,A -85,B 0,C 180,E1 -15439.798,E2 -15439.798} C_VEL
LIN {X 0,Y 312.575,Z 215.549,A -85,B 0,C 180,E1 -15440.873,E2 -15440.873} C_VEL
LIN {X 0,Y 312.484,Z 215.558,A -85,B 0,C 180,E1 -15441.237,E2 -15441.237} C_VEL
LIN {X 0,Y 312.533,Z 215.551,A -85,B 0,C 180,E1 -15444.22,E2 -15444.22} C_VEL
LIN {X 0,Y 312.503,Z 215.559,A -85,B 0,C 180,E1 -15447.334,E2 -15447.334} C_VEL
LIN {X 0,Y 312.509,Z 215.558,A -85,B 0,C 180,E1 -15451.292,E2 -15451.292} C_VEL
LIN {X 0,Y 312.55,Z 215.552,A -85,B 0,C 180,E1 -15454.708,E2 -15454.708} C_VEL
LIN {X 0,Y 312.565,Z 215.548,A -85,B 0,C 180,E1 -15457.527,E2 -15457.527} C_VEL
LIN {X 0,Y 312.591,Z 215.544,A -85,B 0,C 180,E1 -15461.654,E2 -15461.654} C_VEL
LIN {X 0,Y 312.688,Z 215.531,A -85,B 0,C 180,E1 -15465.686,E2 -15465.686} C_VEL
LIN {X 0,Y 312.688,Z 215.53,A -85,B 0,C 180,E1 -15469.641,E2 -15469.641} C_VEL
LIN {X 0,Y 312.799,Z 215.519,A -85,B 0,C 180,E1 -15472.253,E2 -15472.253} C_VEL
LIN {X 0,Y 312.699,Z 215.533,A -85,B 0,C 180,E1 -15474.842,E2 -15474.842} C_VEL
LIN {X 0,Y 312.927,Z 215.502,A -85,B 0,C 180,E1 -15477.426,E2 -15477.426} C_VEL
LIN {X 0,Y 312.982,Z 215.496,A -85,B 0,C 180,E1 -15481.287,E2 -15481.287} C_VEL
LIN {X 0,Y 312.844,Z 215.515,A -85,B 0,C 180,E1 -15486.449,E2 -15486.449} C_VEL
LIN {X 0,Y 312.758,Z 215.522,A -85,B 0,C 180,E1 -15489.05,E2 -15489.05} C_VEL
LIN {X 0,Y 312.627,Z 215.54,A -85,B 0,C 180,E1 -15492.992,E2 -15492.992} C_VEL
LIN {X 0,Y 312.582,Z 215.548,A -85,B 0,C 180,E1 -15495.653,E2 -15495.653} C_VEL
LIN {X 0,Y 312.561,Z 215.552,A -85,B 0,C 180,E1 -15499.711,E2 -15499.711} C_VEL
LIN {X 0,Y 312.519,Z 215.553,A -85,B 0,C 180,E1 -15502.776,E2 -15502.776} C_VEL
LIN {X 0,Y 312.488,Z 215.557,A -85,B 0,C 180,E1 -15506.732,E2 -15506.732} C_VEL
LIN {X 0,Y 312.498,Z 215.561,A -85,B 0,C 180,E1 -15509.655,E2 -15509.655} C_VEL
LIN {X 0,Y 312.522,Z 215.557,A -85,B 0,C 180,E1 -15513.689,E2 -15513.689} C_VEL
LIN {X 0,Y 312.517,Z 215.558,A -85,B 0,C 180,E1 -15517.387,E2 -15517.387} C_VEL
LIN {X 0,Y 312.443,Z 215.564,A -85,B 0,C 180,E1 -15520.717,E2 -15520.717} C_VEL
LIN {X 0,Y 312.452,Z 215.562,A -85,B 0,C 180,E1 -15524.21,E2 -15524.21} C_VEL
LIN {X 0,Y 312.457,Z 215.562,A -85,B 0,C 180,E1 -15527.925,E2 -15527.925} C_VEL
LIN {X 0,Y 312.486,Z 215.558,A -85,B 0,C 180,E1 -15531.922,E2 -15531.922} C_VEL
LIN {X 0,Y 312.535,Z 215.554,A -85,B 0,C 180,E1 -15535.793,E2 -15535.793} C_VEL
LIN {X 0,Y 312.585,Z 215.73,A -85,B 0,C 180,E1 -15536.294,E2 -15536.294} C_VEL
LIN {X 0,Y 315.437,Z 228.829,A -85,B 0,C 180,E1 -15539.779,E2 -15539.779} C_VEL
LIN {X 0,Y 317.263,Z 239.069,A -85,B 0,C 180,E1 -15542.385,E2 -15542.385} C_VEL
LIN {X 0,Y 315.588,Z 253.584,A -85,B 0,C 180,E1 -15545.749,E2 -15545.749} C_VEL
LIN {X 0,Y 320.924,Z 299.147,A -85,B 0,C 180,E1 -15547.316,E2 -15547.316} C_VEL
LIN {X 0,Y 319.337,Z 363.947,A -85,B 0,C 180,E1 -15549.003,E2 -15549.003} C_VEL
LIN {X 0,Y 318.517,Z 376.959,A -85,B 0,C 180,E1 -15549.58,E2 -15549.58} C_VEL
LIN {X 0,Y 317.621,Z 389.138,A -85,B 0,C 180,E1 -15550.363,E2 -15550.363} C_VEL
LIN {X 0,Y 316.356,Z 400.931,A -85,B 0,C 180,E1 -15551.376,E2 -15551.376} C_VEL
LIN {X 0,Y 315.14,Z 412.389,A -85,B 0,C 180,E1 -15552.645,E2 -15552.645} C_VEL
LIN {X 0,Y 313.928,Z 422.752,A -85,B 0,C 180,E1 -15554.083,E2 -15554.083} C_VEL
LIN {X 0,Y 313.146,Z 430.724,A -85,B 0,C 180,E1 -15555.437,E2 -15555.437} C_VEL
LIN {X 0,Y 312.221,Z 439.786,A -85,B 0,C 180,E1 -15557.322,E2 -15557.322} C_VEL
LIN {X 0,Y 311.454,Z 447.307,A -85,B 0,C 180,E1 -15559.271,E2 -15559.271} C_VEL
LIN {X 0,Y 311.174,Z 452.406,A -85,B 0,C 180,E1 -15560.903,E2 -15560.903} C_VEL
LIN {X 0,Y 311.004,Z 457.318,A -85,B 0,C 180,E1 -15562.86,E2 -15562.86} C_VEL
LIN {X 0,Y 311.024,Z 461.042,A -85,B 0,C 180,E1 -15564.814,E2 -15564.814} C_VEL
LIN {X 0,Y 310.985,Z 462.928,A -85,B 0,C 180,E1 -15566.112,E2 -15566.112} C_VEL
LIN {X 0,Y 311.111,Z 464.332,A -85,B 0,C 180,E1 -15567.41,E2 -15567.41} C_VEL
LIN {X 0,Y 311.207,Z 465.293,A -85,B 0,C 180,E1 -15568.706,E2 -15568.706} C_VEL
LIN {X 0,Y 311.207,Z 465.831,A -85,B 0,C 180,E1 -15570,E2 -15570} C_VEL
LIN {X 0,Y 311.177,Z 465.943,A -85,B 0,C 180,E1 -15571.294,E2 -15571.294} C_VEL
LIN {X 0,Y 310.995,Z 465.584,A -85,B 0,C 180,E1 -15572.59,E2 -15572.59} C_VEL
LIN {X 0,Y 310.915,Z 464.822,A -85,B 0,C 180,E1 -15573.888,E2 -15573.888} C_VEL
LIN {X 0,Y 310.826,Z 462.941,A -85,B 0,C 180,E1 -15575.802,E2 -15575.802} C_VEL
LIN {X 0,Y 310.97,Z 459.999,A -85,B 0,C 180,E1 -15577.793,E2 -15577.793} C_VEL
LIN {X 0,Y 311.258,Z 456.063,A -85,B 0,C 180,E1 -15579.749,E2 -15579.749} C_VEL
LIN {X 0,Y 311.833,Z 451,A -85,B 0,C 180,E1 -15581.703,E2 -15581.703} C_VEL
LIN {X 0,Y 313.142,Z 443.501,A -85,B 0,C 180,E1 -15583.961,E2 -15583.961} C_VEL
LIN {X 0,Y 314.391,Z 435.733,A -85,B 0,C 180,E1 -15585.815,E2 -15585.815} C_VEL
LIN {X 0,Y 315.814,Z 427.151,A -85,B 0,C 180,E1 -15587.483,E2 -15587.483} C_VEL
LIN {X 0,Y 317.809,Z 416.147,A -85,B 0,C 180,E1 -15589.204,E2 -15589.204} C_VEL
LIN {X 0,Y 319.731,Z 404.873,A -85,B 0,C 180,E1 -15590.591,E2 -15590.591} C_VEL
LIN {X 0,Y 321.386,Z 393.966,A -85,B 0,C 180,E1 -15591.655,E2 -15591.655} C_VEL
LIN {X 0,Y 323.116,Z 380.998,A -85,B 0,C 180,E1 -15592.626,E2 -15592.626} C_VEL
LIN {X 0,Y 324.491,Z 367.805,A -85,B 0,C 180,E1 -15593.325,E2 -15593.325} C_VEL
LIN {X 0,Y 325.318,Z 354.134,A -85,B 0,C 180,E1 -15593.81,E2 -15593.81} C_VEL
LIN {X 0,Y 327.143,Z 300.152,A -85,B 0,C 180,E1 -15595.235,E2 -15595.235} C_VEL
LIN {X 0,Y 324.73,Z 278.642,A -85,B 0,C 180,E1 -15596.17,E2 -15596.17} C_VEL
LIN {X 0,Y 321.147,Z 258.439,A -85,B 0,C 180,E1 -15597.225,E2 -15597.225} C_VEL
LIN {X 0,Y 319.027,Z 248.085,A -85,B 0,C 180,E1 -15597.861,E2 -15597.861} C_VEL
LIN {X 0,Y 319.435,Z 245.357,A -85,B 0,C 180,E1 -15598.489,E2 -15598.489} C_VEL
LIN {X 0,Y 318.884,Z 240.609,A -85,B 0,C 180,E1 -15599.728,E2 -15599.728} C_VEL
LIN {X 0,Y 316.369,Z 229.15,A -85,B 0,C 180,E1 -15602.987,E2 -15602.987} C_VEL
LIN {X 0,Y 313.498,Z 218.984,A -85,B 0,C 180,E1 -15606.191,E2 -15606.191} C_VEL
LIN {X 0,Y 312.536,Z 215.552,A -85,B 0,C 180,E1 -15607.383,E2 -15607.383} C_VEL
LIN {X 0,Y 312.44,Z 215.563,A -85,B 0,C 180,E1 -15610.717,E2 -15610.717} C_VEL
LIN {X 0,Y 312.451,Z 215.564,A -85,B 0,C 180,E1 -15614.209,E2 -15614.209} C_VEL
LIN {X 0,Y 312.455,Z 215.56,A -85,B 0,C 180,E1 -15617.924,E2 -15617.924} C_VEL
LIN {X 0,Y 312.483,Z 215.558,A -85,B 0,C 180,E1 -15621.922,E2 -15621.922} C_VEL
LIN {X 0,Y 312.53,Z 215.554,A -85,B 0,C 180,E1 -15624.22,E2 -15624.22} C_VEL
LIN {X 0,Y 312.501,Z 215.554,A -85,B 0,C 180,E1 -15627.333,E2 -15627.333} C_VEL
LIN {X 0,Y 312.519,Z 215.553,A -85,B 0,C 180,E1 -15631.287,E2 -15631.287} C_VEL
LIN {X 0,Y 312.551,Z 215.553,A -85,B 0,C 180,E1 -15634.708,E2 -15634.708} C_VEL
LIN {X 0,Y 312.563,Z 215.549,A -85,B 0,C 180,E1 -15637.527,E2 -15637.527} C_VEL
LIN {X 0,Y 312.588,Z 215.546,A -85,B 0,C 180,E1 -15641.653,E2 -15641.653} C_VEL
LIN {X 0,Y 312.685,Z 215.53,A -85,B 0,C 180,E1 -15645.686,E2 -15645.686} C_VEL
LIN {X 0,Y 312.698,Z 215.535,A -85,B 0,C 180,E1 -15649.642,E2 -15649.642} C_VEL
LIN {X 0,Y 312.853,Z 215.515,A -85,B 0,C 180,E1 -15652.254,E2 -15652.254} C_VEL
LIN {X 0,Y 312.714,Z 215.532,A -85,B 0,C 180,E1 -15654.842,E2 -15654.842} C_VEL
LIN {X 0,Y 312.988,Z 215.495,A -85,B 0,C 180,E1 -15658.713,E2 -15658.713} C_VEL
LIN {X 0,Y 312.988,Z 215.498,A -85,B 0,C 180,E1 -15661.287,E2 -15661.287} C_VEL
LIN {X 0,Y 312.707,Z 215.534,A -85,B 0,C 180,E1 -15665.158,E2 -15665.158} C_VEL
LIN {X 0,Y 312.826,Z 215.518,A -85,B 0,C 180,E1 -15667.747,E2 -15667.747} C_VEL
LIN {X 0,Y 312.743,Z 215.595,A -85,B 0,C 180,E1 -15669.458,E2 -15669.458} C_VEL
LIN {X 0,Y 313.707,Z 218.347,A -85,B 0,C 180,E1 -15669.69,E2 -15669.69} C_VEL
LIN {X 0,Y 315.143,Z 220.491,A -85,B 0,C 180,E1 -15669.964,E2 -15669.964} C_VEL
LIN {X 0,Y 322.602,Z 233.71,A -85,B 0,C 180,E1 -15671.381,E2 -15671.381} C_VEL
LIN {X 0,Y 328.923,Z 246.61,A -85,B 0,C 180,E1 -15672.531,E2 -15672.531} C_VEL
LIN {X 0,Y 328.342,Z 264.67,A -85,B 0,C 180,E1 -15673.027,E2 -15673.027} C_VEL
LIN {X 0,Y 326.099,Z 320.57,A -85,B 0,C 180,E1 -15674.534,E2 -15674.534} C_VEL
LIN {X 0,Y 325.429,Z 333.57,A -85,B 0,C 180,E1 -15675.14,E2 -15675.14} C_VEL
LIN {X 0,Y 324.391,Z 345.972,A -85,B 0,C 180,E1 -15675.955,E2 -15675.955} C_VEL
LIN {X 0,Y 323.151,Z 356.668,A -85,B 0,C 180,E1 -15676.879,E2 -15676.879} C_VEL
LIN {X 0,Y 321.655,Z 368.031,A -85,B 0,C 180,E1 -15678.141,E2 -15678.141} C_VEL
LIN {X 0,Y 320.051,Z 378.086,A -85,B 0,C 180,E1 -15679.531,E2 -15679.531} C_VEL
LIN {X 0,Y 318.648,Z 386.555,A -85,B 0,C 180,E1 -15680.98,E2 -15680.98} C_VEL
LIN {X 0,Y 316.994,Z 395.304,A -85,B 0,C 180,E1 -15682.829,E2 -15682.829} C_VEL
LIN {X 0,Y 315.632,Z 401.903,A -85,B 0,C 180,E1 -15684.555,E2 -15684.555} C_VEL
LIN {X 0,Y 314.34,Z 408.097,A -85,B 0,C 180,E1 -15686.58,E2 -15686.58} C_VEL
LIN {X 0,Y 313.148,Z 413.52,A -85,B 0,C 180,E1 -15688.922,E2 -15688.922} C_VEL
LIN {X 0,Y 312.268,Z 417.232,A -85,B 0,C 180,E1 -15691.214,E2 -15691.214} C_VEL
LIN {X 0,Y 311.601,Z 419.524,A -85,B 0,C 180,E1 -15693.435,E2 -15693.435} C_VEL
LIN {X 0,Y 311.152,Z 420.636,A -85,B 0,C 180,E1 -15695.963,E2 -15695.963} C_VEL
LIN {X 0,Y 311.02,Z 420.488,A -85,B 0,C 180,E1 -15697.732,E2 -15697.732} C_VEL
LIN {X 0,Y 311.023,Z 419.346,A -85,B 0,C 180,E1 -15699.801,E2 -15699.801} C_VEL
LIN {X 0,Y 311.221,Z 417.202,A -85,B 0,C 180,E1 -15701.824,E2 -15701.824} C_VEL
LIN {X 0,Y 311.676,Z 412.996,A -85,B 0,C 180,E1 -15704.348,E2 -15704.348} C_VEL
LIN {X 0,Y 312.093,Z 409.005,A -85,B 0,C 180,E1 -15706.105,E2 -15706.105} C_VEL
LIN {X 0,Y 312.76,Z 402.703,A -85,B 0,C 180,E1 -15708.267,E2 -15708.267} C_VEL
LIN {X 0,Y 313.47,Z 396.089,A -85,B 0,C 180,E1 -15710.071,E2 -15710.071} C_VEL
LIN {X 0,Y 314.449,Z 388.269,A -85,B 0,C 180,E1 -15711.803,E2 -15711.803} C_VEL
LIN {X 0,Y 315.536,Z 378.206,A -85,B 0,C 180,E1 -15713.6,E2 -15713.6} C_VEL
LIN {X 0,Y 316.549,Z 368.414,A -85,B 0,C 180,E1 -15715.015,E2 -15715.015} C_VEL
LIN {X 0,Y 317.611,Z 357.184,A -85,B 0,C 180,E1 -15716.319,E2 -15716.319} C_VEL
LIN {X 0,Y 318.578,Z 345.179,A -85,B 0,C 180,E1 -15717.407,E2 -15717.407} C_VEL
LIN {X 0,Y 319.396,Z 332.286,A -85,B 0,C 180,E1 -15718.29,E2 -15718.29} C_VEL
LIN {X 0,Y 319.85,Z 320.426,A -85,B 0,C 180,E1 -15718.866,E2 -15718.866} C_VEL
LIN {X 0,Y 320.311,Z 302.326,A -85,B 0,C 180,E1 -15719.396,E2 -15719.396} C_VEL
LIN {X 0,Y 321.836,Z 240.045,A -85,B 0,C 180,E1 -15720.977,E2 -15720.977} C_VEL
LIN {X 0,Y 312.731,Z 216.361,A -85,B 0,C 180,E1 -15722.205,E2 -15722.205} C_VEL
LIN {X 0,Y 312.586,Z 215.579,A -85,B 0,C 180,E1 -15722.237,E2 -15722.237} C_VEL
LIN {X 0,Y 312.585,Z 215.548,A -85,B 0,C 180,E1 -15724.711,E2 -15724.711} C_VEL
LIN {X 0,Y 312.564,Z 215.549,A -85,B 0,C 180,E1 -15727.528,E2 -15727.528} C_VEL
LIN {X 0,Y 312.589,Z 215.545,A -85,B 0,C 180,E1 -15731.654,E2 -15731.654} C_VEL
LIN {X 0,Y 312.686,Z 215.533,A -85,B 0,C 180,E1 -15735.686,E2 -15735.686} C_VEL
LIN {X 0,Y 312.686,Z 215.533,A -85,B 0,C 180,E1 -15739.642,E2 -15739.642} C_VEL
LIN {X 0,Y 312.8,Z 215.52,A -85,B 0,C 180,E1 -15742.253,E2 -15742.253} C_VEL
LIN {X 0,Y 312.703,Z 215.534,A -85,B 0,C 180,E1 -15744.842,E2 -15744.842} C_VEL
LIN {X 0,Y 312.933,Z 215.502,A -85,B 0,C 180,E1 -15747.426,E2 -15747.426} C_VEL
LIN {X 0,Y 313.068,Z 215.486,A -85,B 0,C 180,E1 -15750,E2 -15750} C_VEL
LIN {X 0,Y 312.924,Z 215.507,A -85,B 0,C 180,E1 -15752.575,E2 -15752.575} C_VEL
LIN {X 0,Y 312.853,Z 215.516,A -85,B 0,C 180,E1 -15756.45,E2 -15756.45} C_VEL
LIN {X 0,Y 312.756,Z 215.524,A -85,B 0,C 180,E1 -15759.05,E2 -15759.05} C_VEL
LIN {X 0,Y 312.636,Z 215.539,A -85,B 0,C 180,E1 -15762.991,E2 -15762.991} C_VEL
LIN {X 0,Y 312.64,Z 215.54,A -85,B 0,C 180,E1 -15765.65,E2 -15765.65} C_VEL
LIN {X 0,Y 312.611,Z 215.542,A -85,B 0,C 180,E1 -15769.226,E2 -15769.226} C_VEL
LIN {X 0,Y 312.526,Z 215.552,A -85,B 0,C 180,E1 -15772.78,E2 -15772.78} C_VEL
LIN {X 0,Y 312.537,Z 215.556,A -85,B 0,C 180,E1 -15775.91,E2 -15775.91} C_VEL
LIN {X 0,Y 312.502,Z 215.56,A -85,B 0,C 180,E1 -15779.655,E2 -15779.655} C_VEL
LIN {X 0,Y 312.521,Z 215.558,A -85,B 0,C 180,E1 -15783.689,E2 -15783.689} C_VEL
LIN {X 0,Y 312.517,Z 215.555,A -85,B 0,C 180,E1 -15787.387,E2 -15787.387} C_VEL
LIN {X 0,Y 312.49,Z 215.556,A -85,B 0,C 180,E1 -15790.71,E2 -15790.71} C_VEL
LIN {X 0,Y 312.453,Z 215.562,A -85,B 0,C 180,E1 -15794.21,E2 -15794.21} C_VEL
LIN {X 0,Y 312.457,Z 215.562,A -85,B 0,C 180,E1 -15797.925,E2 -15797.925} C_VEL
LIN {X 0,Y 312.484,Z 215.558,A -85,B 0,C 180,E1 -15801.237,E2 -15801.237} C_VEL
LIN {X 0,Y 311.809,Z 215.642,A -85,B 0,C 180,E1 -15802.313,E2 -15802.313} C_VEL
LIN {X 0,Y 308.981,Z 215.993,A -85,B 0,C 180,E1 -15804.067,E2 -15804.067} C_VEL
LIN {X 0,Y 306.579,Z 216.296,A -85,B 0,C 180,E1 -15805.488,E2 -15805.488} C_VEL
LIN {X 0,Y 305.53,Z 216.425,A -85,B 0,C 180,E1 -15806.588,E2 -15806.588} C_VEL
LIN {X 0,Y 305.434,Z 216.433,A -85,B 0,C 180,E1 -15806.96,E2 -15806.96} C_VEL
LIN {X 0,Y 305.478,Z 216.435,A -85,B 0,C 180,E1 -15811.109,E2 -15811.109} C_VEL
LIN {X 0,Y 305.502,Z 216.426,A -85,B 0,C 180,E1 -15814.082,E2 -15814.082} C_VEL
LIN {X 0,Y 305.478,Z 216.432,A -85,B 0,C 180,E1 -15818.401,E2 -15818.401} C_VEL
LIN {X 0,Y 305.55,Z 216.423,A -85,B 0,C 180,E1 -15821.215,E2 -15821.215} C_VEL
LIN {X 0,Y 305.629,Z 216.411,A -85,B 0,C 180,E1 -15825.348,E2 -15825.348} C_VEL
LIN {X 0,Y 305.627,Z 216.408,A -85,B 0,C 180,E1 -15829.399,E2 -15829.399} C_VEL
LIN {X 0,Y 305.749,Z 216.395,A -85,B 0,C 180,E1 -15832.073,E2 -15832.073} C_VEL
LIN {X 0,Y 305.668,Z 216.409,A -85,B 0,C 180,E1 -15834.723,E2 -15834.723} C_VEL
LIN {X 0,Y 305.942,Z 216.375,A -85,B 0,C 180,E1 -15838.684,E2 -15838.684} C_VEL
LIN {X 0,Y 305.948,Z 216.372,A -85,B 0,C 180,E1 -15841.316,E2 -15841.316} C_VEL
LIN {X 0,Y 305.789,Z 216.391,A -85,B 0,C 180,E1 -15846.599,E2 -15846.599} C_VEL
LIN {X 0,Y 305.701,Z 216.401,A -85,B 0,C 180,E1 -15849.261,E2 -15849.261} C_VEL
LIN {X 0,Y 305.575,Z 216.419,A -85,B 0,C 180,E1 -15853.297,E2 -15853.297} C_VEL
LIN {X 0,Y 305.535,Z 216.425,A -85,B 0,C 180,E1 -15857.399,E2 -15857.399} C_VEL
LIN {X 0,Y 305.497,Z 216.429,A -85,B 0,C 180,E1 -15860.187,E2 -15860.187} C_VEL
LIN {X 0,Y 305.458,Z 216.434,A -85,B 0,C 180,E1 -15864.466,E2 -15864.466} C_VEL
LIN {X 0,Y 305.454,Z 216.436,A -85,B 0,C 180,E1 -15867.398,E2 -15867.398} C_VEL
LIN {X 0,Y 305.432,Z 216.435,A -85,B 0,C 180,E1 -15870.413,E2 -15870.413} C_VEL
LIN {X 0,Y 305.467,Z 216.433,A -85,B 0,C 180,E1 -15874.078,E2 -15874.078} C_VEL
LIN {X 0,Y 305.456,Z 216.434,A -85,B 0,C 180,E1 -15876.742,E2 -15876.742} C_VEL
LIN {X 0,Y 305.411,Z 216.439,A -85,B 0,C 180,E1 -15880.59,E2 -15880.59} C_VEL
LIN {X 0,Y 305.423,Z 216.44,A -85,B 0,C 180,E1 -15883.656,E2 -15883.656} C_VEL
LIN {X 0,Y 305.437,Z 216.439,A -85,B 0,C 180,E1 -15887.418,E2 -15887.418} C_VEL
LIN {X 0,Y 305.462,Z 216.435,A -85,B 0,C 180,E1 -15891.595,E2 -15891.595} C_VEL
LIN {X 0,Y 305.516,Z 216.464,A -85,B 0,C 180,E1 -15895.908,E2 -15895.908} C_VEL
LIN {X 0,Y 308.392,Z 229.767,A -85,B 0,C 180,E1 -15899.532,E2 -15899.532} C_VEL
LIN {X 0,Y 310.213,Z 239.502,A -85,B 0,C 180,E1 -15902.075,E2 -15902.075} C_VEL
LIN {X 0,Y 308.985,Z 250.596,A -85,B 0,C 180,E1 -15904.719,E2 -15904.719} C_VEL
LIN {X 0,Y 308.702,Z 253.05,A -85,B 0,C 180,E1 -15905.303,E2 -15905.303} C_VEL
LIN {X 0,Y 314.149,Z 300.719,A -85,B 0,C 180,E1 -15906.977,E2 -15906.977} C_VEL
LIN {X 0,Y 312.519,Z 363.515,A -85,B 0,C 180,E1 -15908.652,E2 -15908.652} C_VEL
LIN {X 0,Y 311.629,Z 377.224,A -85,B 0,C 180,E1 -15909.28,E2 -15909.28} C_VEL
LIN {X 0,Y 310.585,Z 390.136,A -85,B 0,C 180,E1 -15910.158,E2 -15910.158} C_VEL
LIN {X 0,Y 309.316,Z 402.433,A -85,B 0,C 180,E1 -15911.28,E2 -15911.28} C_VEL
LIN {X 0,Y 307.964,Z 413.485,A -85,B 0,C 180,E1 -15912.571,E2 -15912.571} C_VEL
LIN {X 0,Y 306.802,Z 423.498,A -85,B 0,C 180,E1 -15914.044,E2 -15914.044} C_VEL
LIN {X 0,Y 305.888,Z 432.634,A -85,B 0,C 180,E1 -15915.7,E2 -15915.7} C_VEL
LIN {X 0,Y 304.962,Z 441.522,A -85,B 0,C 180,E1 -15917.691,E2 -15917.691} C_VEL
LIN {X 0,Y 304.29,Z 448.573,A -85,B 0,C 180,E1 -15919.688,E2 -15919.688} C_VEL
LIN {X 0,Y 303.973,Z 455.031,A -85,B 0,C 180,E1 -15922.026,E2 -15922.026} C_VEL
LIN {X 0,Y 303.955,Z 458.875,A -85,B 0,C 180,E1 -15923.85,E2 -15923.85} C_VEL
LIN {X 0,Y 303.913,Z 462.248,A -85,B 0,C 180,E1 -15926.022,E2 -15926.022} C_VEL
LIN {X 0,Y 304.018,Z 463.706,A -85,B 0,C 180,E1 -15927.35,E2 -15927.35} C_VEL
LIN {X 0,Y 304.146,Z 464.695,A -85,B 0,C 180,E1 -15928.676,E2 -15928.676} C_VEL
LIN {X 0,Y 304.147,Z 465.258,A -85,B 0,C 180,E1 -15930,E2 -15930} C_VEL
LIN {X 0,Y 304.113,Z 465.406,A -85,B 0,C 180,E1 -15931.324,E2 -15931.324} C_VEL
LIN {X 0,Y 303.901,Z 465.089,A -85,B 0,C 180,E1 -15932.651,E2 -15932.651} C_VEL
LIN {X 0,Y 303.836,Z 464.357,A -85,B 0,C 180,E1 -15933.979,E2 -15933.979} C_VEL
LIN {X 0,Y 303.73,Z 462.77,A -85,B 0,C 180,E1 -15935.744,E2 -15935.744} C_VEL
LIN {X 0,Y 303.906,Z 459.65,A -85,B 0,C 180,E1 -15937.975,E2 -15937.975} C_VEL
LIN {X 0,Y 304.234,Z 455.774,A -85,B 0,C 180,E1 -15939.977,E2 -15939.977} C_VEL
LIN {X 0,Y 304.853,Z 450.772,A -85,B 0,C 180,E1 -15941.975,E2 -15941.975} C_VEL
LIN {X 0,Y 306.212,Z 443.356,A -85,B 0,C 180,E1 -15944.284,E2 -15944.284} C_VEL
LIN {X 0,Y 307.606,Z 434.994,A -85,B 0,C 180,E1 -15946.343,E2 -15946.343} C_VEL
LIN {X 0,Y 309.417,Z 425.495,A -85,B 0,C 180,E1 -15948.198,E2 -15948.198} C_VEL
LIN {X 0,Y 311.339,Z 415.356,A -85,B 0,C 180,E1 -15949.791,E2 -15949.791} C_VEL
LIN {X 0,Y 313.311,Z 404.016,A -85,B 0,C 180,E1 -15951.205,E2 -15951.205} C_VEL
LIN {X 0,Y 315.355,Z 391.288,A -85,B 0,C 180,E1 -15952.435,E2 -15952.435} C_VEL
LIN {X 0,Y 317.038,Z 378.701,A -85,B 0,C 180,E1 -15953.343,E2 -15953.343} C_VEL
LIN {X 0,Y 318.481,Z 364.929,A -85,B 0,C 180,E1 -15954.051,E2 -15954.051} C_VEL
LIN {X 0,Y 319.266,Z 351.321,A -85,B 0,C 180,E1 -15954.507,E2 -15954.507} C_VEL
LIN {X 0,Y 321.119,Z 301.34,A -85,B 0,C 180,E1 -15955.859,E2 -15955.859} C_VEL
LIN {X 0,Y 318.688,Z 279.431,A -85,B 0,C 180,E1 -15956.843,E2 -15956.843} C_VEL
LIN {X 0,Y 315.079,Z 258.786,A -85,B 0,C 180,E1 -15957.971,E2 -15957.971} C_VEL
